KUKA KRL program: EPS_2_251112_SAMH04_A_20250918124117.src

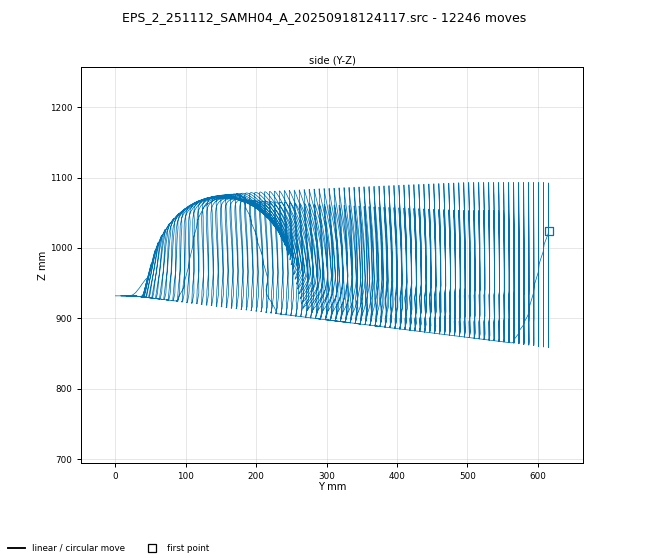
[picture p0: tool path of EPS_2_251112_SAMH04_A_20250918124117.src, 12246 of 12248 moves have a stored position in this frame; points joined in program order, loops and branches not executed]
&ACCESS RVP
&REL 4
&COMMENT QRS 19112012
&PARAM EDITMASK = *
DEF PART()
EXT BAS (BAS_COMMAND :IN,REAL :IN )
INT I
BAS (#INITMOV,0 )

;KUKA QRS Post kuka4.cps  Date:22-06-2017 !

File_ID=2836

QRS_PRE_INIT()

;Init var - Until changes are made in qrs_pre_init
Outlet_Square_prg=0
Inlet_1_Square_prg=0
Inlet_2_Square_prg=0
Inlet_3_Square_prg=0
Inlet_4_Square_prg=0
Inlet_5_Square_prg=0

Outlet_1={X 0.000, Y 497.840, Z 1018.000, B 0.000, E1 0.000 }
Inlet_1={X 0.000, Y 500.690, Z 978.000, B 0.000, E1 90.000 }
Outlet_1_type=150
Inlet_1_type=150
;QRS#1=Sidecore dimensions
;QRS#2=150-6" PVC SDR 28
;QRS#3=150-6" PVC SDR 28
;QRS#4=
;QRS#5=
;QRS#6=
;QRS#7=
;QRS#8=
;QRS#9=10-06 PSX
;QRS#10=10-06 PSX
;QRS#11=
;QRS#12=
;QRS#13=
;QRS#14=
;QRS#15=
;QRS#16=1220x127x1372 4,5'
;QRS#17=EPS Height
;QRS#18=1093
;QRS#19=*
;QRS#20= UPDATED VERSION 22-06-2017
;QRS#21=*
Outlet_Square=070
Inlet_1_Square=070
Inlet_2_Square=0
Inlet_3_Square=0
Inlet_4_Square=0
Inlet_5_Square=0
Mill_Square=1
Outlet_Square_Prg=203
Inlet_1_Square_prg=203

QRS_INIT()

$ADVANCE=5

; T1
PTP {E1 173.415,E2 173.415}
PTP {X 0,Y 615.497,A -85,B 0,C 180,E1 173.415,E2 173.415,E3 0,E4 0,E5 0,E6 0}
QRS_SPEED_INIT()
LIN {X 0,Y 615.497,Z 1023.816,A -85,B 0,C 180,E1 173.415,E2 173.415,E3 0,E4 0,E5 0,E6 0} C_VEL
LIN {X 0,Y 615.483,Z 1015.551,A -85,B 0,C 180,E1 172.702,E2 172.702} C_VEL
LIN {X 0,Y 615.494,Z 1005.669,A -85,B 0,C 180,E1 172.042,E2 172.042} C_VEL
LIN {X 0,Y 615.492,Z 997.912,A -85,B 0,C 180,E1 171.628,E2 171.628} C_VEL
LIN {X 0,Y 615.46,Z 989.058,A -85,B 0,C 180,E1 171.256,E2 171.256} C_VEL
LIN {X 0,Y 615.451,Z 979.837,A -85,B 0,C 180,E1 170.966,E2 170.966} C_VEL
LIN {X 0,Y 615.452,Z 970.156,A -85,B 0,C 180,E1 170.759,E2 170.759} C_VEL
LIN {X 0,Y 615.49,Z 894.306,A -85,B 0,C 180,E1 169.847,E2 169.847} C_VEL
LIN {X 0,Y 615.486,Z 880.811,A -85,B 0,C 180,E1 167.134,E2 167.134} C_VEL
LIN {X 0,Y 615.453,Z 867.509,A -85,B 0,C 180,E1 164.433,E2 164.433} C_VEL
LIN {X 0,Y 615.432,Z 858.511,A -85,B 0,C 180,E1 162.556,E2 162.556} C_VEL
LIN {X 0,Y 615.415,Z 858.509,A -85,B 0,C 180,E1 159.964,E2 159.964} C_VEL
LIN {X 0,Y 615.466,Z 858.507,A -85,B 0,C 180,E1 157.154,E2 157.154} C_VEL
LIN {X 0,Y 615.441,Z 858.511,A -85,B 0,C 180,E1 154.282,E2 154.282} C_VEL
LIN {X 0,Y 615.431,Z 858.511,A -85,B 0,C 180,E1 152.082,E2 152.082} C_VEL
LIN {X 0,Y 615.419,Z 858.51,A -85,B 0,C 180,E1 149.836,E2 149.836} C_VEL
LIN {X 0,Y 615.412,Z 858.51,A -85,B 0,C 180,E1 147.538,E2 147.538} C_VEL
LIN {X 0,Y 615.447,Z 858.511,A -85,B 0,C 180,E1 145.975,E2 145.975} C_VEL
LIN {X 0,Y 615.421,Z 858.51,A -85,B 0,C 180,E1 143.57,E2 143.57} C_VEL
LIN {X 0,Y 615.415,Z 858.509,A -85,B 0,C 180,E1 141.09,E2 141.09} C_VEL
LIN {X 0,Y 615.417,Z 858.508,A -85,B 0,C 180,E1 138.913,E2 138.913} C_VEL
LIN {X 0,Y 615.42,Z 858.508,A -85,B 0,C 180,E1 136.749,E2 136.749} C_VEL
LIN {X 0,Y 615.469,Z 858.506,A -85,B 0,C 180,E1 134.151,E2 134.151} C_VEL
LIN {X 0,Y 615.462,Z 858.513,A -85,B 0,C 180,E1 131.476,E2 131.476} C_VEL
LIN {X 0,Y 615.419,Z 858.51,A -85,B 0,C 180,E1 128.91,E2 128.91} C_VEL
LIN {X 0,Y 615.415,Z 858.509,A -85,B 0,C 180,E1 126.43,E2 126.43} C_VEL
LIN {X 0,Y 615.431,Z 858.508,A -85,B 0,C 180,E1 124.026,E2 124.026} C_VEL
LIN {X 0,Y 615.476,Z 858.512,A -85,B 0,C 180,E1 121.083,E2 121.083} C_VEL
LIN {X 0,Y 615.42,Z 858.51,A -85,B 0,C 180,E1 118.438,E2 118.438} C_VEL
LIN {X 0,Y 615.423,Z 858.511,A -85,B 0,C 180,E1 116.447,E2 116.447} C_VEL
LIN {X 0,Y 615.421,Z 858.51,A -85,B 0,C 180,E1 114.275,E2 114.275} C_VEL
LIN {X 0,Y 615.419,Z 858.51,A -85,B 0,C 180,E1 112.139,E2 112.139} C_VEL
LIN {X 0,Y 615.418,Z 858.51,A -85,B 0,C 180,E1 110.035,E2 110.035} C_VEL
LIN {X 0,Y 615.419,Z 858.51,A -85,B 0,C 180,E1 107.959,E2 107.959} C_VEL
LIN {X 0,Y 615.421,Z 858.51,A -85,B 0,C 180,E1 105.907,E2 105.907} C_VEL
LIN {X 0,Y 615.425,Z 858.51,A -85,B 0,C 180,E1 103.876,E2 103.876} C_VEL
LIN {X 0,Y 615.43,Z 858.511,A -85,B 0,C 180,E1 101.862,E2 101.862} C_VEL
LIN {X 0,Y 615.439,Z 858.511,A -85,B 0,C 180,E1 99.863,E2 99.863} C_VEL
LIN {X 0,Y 615.45,Z 858.511,A -85,B 0,C 180,E1 97.876,E2 97.876} C_VEL
LIN {X 0,Y 615.414,Z 858.51,A -85,B 0,C 180,E1 95.242,E2 95.242} C_VEL
LIN {X 0,Y 615.417,Z 858.51,A -85,B 0,C 180,E1 93.273,E2 93.273} C_VEL
LIN {X 0,Y 615.42,Z 858.511,A -85,B 0,C 180,E1 91.309,E2 91.309} C_VEL
LIN {X 0,Y 615.432,Z 858.511,A -85,B 0,C 180,E1 89.346,E2 89.346} C_VEL
LIN {X 0,Y 615.446,Z 858.511,A -85,B 0,C 180,E1 87.382,E2 87.382} C_VEL
LIN {X 0,Y 615.413,Z 858.51,A -85,B 0,C 180,E1 84.758,E2 84.758} C_VEL
LIN {X 0,Y 615.416,Z 858.51,A -85,B 0,C 180,E1 82.783,E2 82.783} C_VEL
LIN {X 0,Y 615.421,Z 858.51,A -85,B 0,C 180,E1 80.8,E2 80.8} C_VEL
LIN {X 0,Y 615.427,Z 858.511,A -85,B 0,C 180,E1 78.806,E2 78.806} C_VEL
LIN {X 0,Y 615.434,Z 858.511,A -85,B 0,C 180,E1 76.797,E2 76.797} C_VEL
LIN {X 0,Y 615.437,Z 858.512,A -85,B 0,C 180,E1 74.772,E2 74.772} C_VEL
LIN {X 0,Y 615.446,Z 858.511,A -85,B 0,C 180,E1 72.728,E2 72.728} C_VEL
LIN {X 0,Y 615.448,Z 858.511,A -85,B 0,C 180,E1 70.661,E2 70.661} C_VEL
LIN {X 0,Y 615.448,Z 858.511,A -85,B 0,C 180,E1 68.566,E2 68.566} C_VEL
LIN {X 0,Y 615.414,Z 858.51,A -85,B 0,C 180,E1 66.008,E2 66.008} C_VEL
LIN {X 0,Y 615.437,Z 858.511,A -85,B 0,C 180,E1 64.282,E2 64.282} C_VEL
LIN {X 0,Y 615.428,Z 858.511,A -85,B 0,C 180,E1 62.082,E2 62.082} C_VEL
LIN {X 0,Y 615.418,Z 858.51,A -85,B 0,C 180,E1 59.836,E2 59.836} C_VEL
LIN {X 0,Y 615.41,Z 858.51,A -85,B 0,C 180,E1 57.538,E2 57.538} C_VEL
LIN {X 0,Y 615.444,Z 858.511,A -85,B 0,C 180,E1 55.975,E2 55.975} C_VEL
LIN {X 0,Y 615.419,Z 858.51,A -85,B 0,C 180,E1 53.57,E2 53.57} C_VEL
LIN {X 0,Y 615.411,Z 858.51,A -85,B 0,C 180,E1 51.09,E2 51.09} C_VEL
LIN {X 0,Y 615.416,Z 858.509,A -85,B 0,C 180,E1 48.914,E2 48.914} C_VEL
LIN {X 0,Y 615.419,Z 858.509,A -85,B 0,C 180,E1 46.749,E2 46.749} C_VEL
LIN {X 0,Y 615.468,Z 858.507,A -85,B 0,C 180,E1 44.152,E2 44.152} C_VEL
LIN {X 0,Y 615.462,Z 858.512,A -85,B 0,C 180,E1 41.477,E2 41.477} C_VEL
LIN {X 0,Y 615.426,Z 858.511,A -85,B 0,C 180,E1 39.055,E2 39.055} C_VEL
LIN {X 0,Y 615.413,Z 858.509,A -85,B 0,C 180,E1 36.43,E2 36.43} C_VEL
LIN {X 0,Y 615.43,Z 858.508,A -85,B 0,C 180,E1 34.026,E2 34.026} C_VEL
LIN {X 0,Y 615.455,Z 858.508,A -85,B 0,C 180,E1 31.688,E2 31.688} C_VEL
LIN {X 0,Y 615.433,Z 858.511,A -85,B 0,C 180,E1 28.661,E2 28.661} C_VEL
LIN {X 0,Y 615.423,Z 858.511,A -85,B 0,C 180,E1 26.448,E2 26.448} C_VEL
LIN {X 0,Y 615.418,Z 858.51,A -85,B 0,C 180,E1 24.275,E2 24.275} C_VEL
LIN {X 0,Y 615.416,Z 858.51,A -85,B 0,C 180,E1 22.14,E2 22.14} C_VEL
LIN {X 0,Y 615.415,Z 858.511,A -85,B 0,C 180,E1 20.036,E2 20.036} C_VEL
LIN {X 0,Y 615.416,Z 858.51,A -85,B 0,C 180,E1 17.959,E2 17.959} C_VEL
LIN {X 0,Y 615.418,Z 858.51,A -85,B 0,C 180,E1 15.907,E2 15.907} C_VEL
LIN {X 0,Y 615.422,Z 858.511,A -85,B 0,C 180,E1 13.876,E2 13.876} C_VEL
LIN {X 0,Y 615.427,Z 858.511,A -85,B 0,C 180,E1 11.862,E2 11.862} C_VEL
LIN {X 0,Y 615.436,Z 858.511,A -85,B 0,C 180,E1 9.863,E2 9.863} C_VEL
LIN {X 0,Y 615.447,Z 858.511,A -85,B 0,C 180,E1 7.876,E2 7.876} C_VEL
LIN {X 0,Y 615.411,Z 858.51,A -85,B 0,C 180,E1 5.242,E2 5.242} C_VEL
LIN {X 0,Y 615.412,Z 858.511,A -85,B 0,C 180,E1 3.274,E2 3.274} C_VEL
LIN {X 0,Y 615.421,Z 858.511,A -85,B 0,C 180,E1 1.309,E2 1.309} C_VEL
LIN {X 0,Y 615.431,Z 858.511,A -85,B 0,C 180,E1 -0.654,E2 -0.654} C_VEL
LIN {X 0,Y 615.443,Z 858.511,A -85,B 0,C 180,E1 -2.618,E2 -2.618} C_VEL
LIN {X 0,Y 615.411,Z 858.51,A -85,B 0,C 180,E1 -5.242,E2 -5.242} C_VEL
LIN {X 0,Y 615.414,Z 858.51,A -85,B 0,C 180,E1 -7.216,E2 -7.216} C_VEL
LIN {X 0,Y 615.418,Z 858.511,A -85,B 0,C 180,E1 -9.2,E2 -9.2} C_VEL
LIN {X 0,Y 615.424,Z 858.511,A -85,B 0,C 180,E1 -11.194,E2 -11.194} C_VEL
LIN {X 0,Y 615.431,Z 858.511,A -85,B 0,C 180,E1 -13.202,E2 -13.202} C_VEL
LIN {X 0,Y 615.437,Z 858.511,A -85,B 0,C 180,E1 -15.227,E2 -15.227} C_VEL
LIN {X 0,Y 615.442,Z 858.511,A -85,B 0,C 180,E1 -17.272,E2 -17.272} C_VEL
LIN {X 0,Y 615.445,Z 858.512,A -85,B 0,C 180,E1 -19.339,E2 -19.339} C_VEL
LIN {X 0,Y 615.445,Z 858.512,A -85,B 0,C 180,E1 -21.433,E2 -21.433} C_VEL
LIN {X 0,Y 615.412,Z 858.51,A -85,B 0,C 180,E1 -23.992,E2 -23.992} C_VEL
LIN {X 0,Y 615.434,Z 858.511,A -85,B 0,C 180,E1 -25.718,E2 -25.718} C_VEL
LIN {X 0,Y 615.425,Z 858.511,A -85,B 0,C 180,E1 -27.918,E2 -27.918} C_VEL
LIN {X 0,Y 615.416,Z 858.511,A -85,B 0,C 180,E1 -30.164,E2 -30.164} C_VEL
LIN {X 0,Y 615.408,Z 858.51,A -85,B 0,C 180,E1 -32.462,E2 -32.462} C_VEL
LIN {X 0,Y 615.441,Z 858.511,A -85,B 0,C 180,E1 -34.025,E2 -34.025} C_VEL
LIN {X 0,Y 615.416,Z 858.511,A -85,B 0,C 180,E1 -36.429,E2 -36.429} C_VEL
LIN {X 0,Y 615.411,Z 858.51,A -85,B 0,C 180,E1 -38.91,E2 -38.91} C_VEL
LIN {X 0,Y 615.414,Z 858.509,A -85,B 0,C 180,E1 -41.086,E2 -41.086} C_VEL
LIN {X 0,Y 615.417,Z 858.509,A -85,B 0,C 180,E1 -43.251,E2 -43.251} C_VEL
LIN {X 0,Y 615.468,Z 858.508,A -85,B 0,C 180,E1 -45.848,E2 -45.848} C_VEL
LIN {X 0,Y 615.459,Z 858.512,A -85,B 0,C 180,E1 -48.523,E2 -48.523} C_VEL
LIN {X 0,Y 615.423,Z 858.511,A -85,B 0,C 180,E1 -50.945,E2 -50.945} C_VEL
LIN {X 0,Y 615.411,Z 858.51,A -85,B 0,C 180,E1 -53.57,E2 -53.57} C_VEL
LIN {X 0,Y 615.428,Z 858.509,A -85,B 0,C 180,E1 -55.974,E2 -55.974} C_VEL
LIN {X 0,Y 615.469,Z 858.512,A -85,B 0,C 180,E1 -58.917,E2 -58.917} C_VEL
LIN {X 0,Y 615.415,Z 858.511,A -85,B 0,C 180,E1 -61.562,E2 -61.562} C_VEL
LIN {X 0,Y 615.42,Z 858.511,A -85,B 0,C 180,E1 -63.553,E2 -63.553} C_VEL
LIN {X 0,Y 615.416,Z 858.511,A -85,B 0,C 180,E1 -65.725,E2 -65.725} C_VEL
LIN {X 0,Y 615.414,Z 858.511,A -85,B 0,C 180,E1 -67.861,E2 -67.861} C_VEL
LIN {X 0,Y 615.431,Z 858.559,A -85,B 0,C 180,E1 -68.566,E2 -68.566} C_VEL
LIN {X 0,Y 615.473,Z 876.687,A -85,B 0,C 180,E1 -71.399,E2 -71.399} C_VEL
LIN {X 0,Y 615.484,Z 894.205,A -85,B 0,C 180,E1 -74.095,E2 -74.095} C_VEL
LIN {X 0,Y 615.455,Z 912.003,A -85,B 0,C 180,E1 -76.798,E2 -76.798} C_VEL
LIN {X 0,Y 615.493,Z 930.889,A -85,B 0,C 180,E1 -79.639,E2 -79.639} C_VEL
LIN {X 0,Y 615.483,Z 932.416,A -85,B 0,C 180,E1 -79.868,E2 -79.868} C_VEL
LIN {X 0,Y 615.47,Z 1009.935,A -85,B 0,C 180,E1 -80.801,E2 -80.801} C_VEL
LIN {X 0,Y 615.465,Z 1019.696,A -85,B 0,C 180,E1 -81.008,E2 -81.008} C_VEL
LIN {X 0,Y 615.471,Z 1030.154,A -85,B 0,C 180,E1 -81.339,E2 -81.339} C_VEL
LIN {X 0,Y 615.497,Z 1040.424,A -85,B 0,C 180,E1 -81.794,E2 -81.794} C_VEL
LIN {X 0,Y 615.477,Z 1050.199,A -85,B 0,C 180,E1 -82.372,E2 -82.372} C_VEL
LIN {X 0,Y 615.493,Z 1057.933,A -85,B 0,C 180,E1 -82.942,E2 -82.942} C_VEL
LIN {X 0,Y 615.497,Z 1065.332,A -85,B 0,C 180,E1 -83.608,E2 -83.608} C_VEL
LIN {X 0,Y 615.498,Z 1072.736,A -85,B 0,C 180,E1 -84.43,E2 -84.43} C_VEL
LIN {X 0,Y 615.497,Z 1078.532,A -85,B 0,C 180,E1 -85.251,E2 -85.251} C_VEL
LIN {X 0,Y 615.493,Z 1083.1,A -85,B 0,C 180,E1 -86.071,E2 -86.071} C_VEL
LIN {X 0,Y 615.493,Z 1086.068,A -85,B 0,C 180,E1 -86.727,E2 -86.727} C_VEL
LIN {X 0,Y 615.494,Z 1088.356,A -85,B 0,C 180,E1 -87.382,E2 -87.382} C_VEL
LIN {X 0,Y 615.499,Z 1090.085,A -85,B 0,C 180,E1 -88.037,E2 -88.037} C_VEL
LIN {X 0,Y 615.493,Z 1091.33,A -85,B 0,C 180,E1 -88.691,E2 -88.691} C_VEL
LIN {X 0,Y 615.491,Z 1092.104,A -85,B 0,C 180,E1 -89.346,E2 -89.346} C_VEL
LIN {X 0,Y 615.491,Z 1092.389,A -85,B 0,C 180,E1 -90,E2 -90} C_VEL
LIN {X 0,Y 615.491,Z 1092.104,A -85,B 0,C 180,E1 -90.654,E2 -90.654} C_VEL
LIN {X 0,Y 615.493,Z 1091.33,A -85,B 0,C 180,E1 -91.308,E2 -91.308} C_VEL
LIN {X 0,Y 615.499,Z 1090.085,A -85,B 0,C 180,E1 -91.963,E2 -91.963} C_VEL
LIN {X 0,Y 615.488,Z 1087.221,A -85,B 0,C 180,E1 -92.945,E2 -92.945} C_VEL
LIN {X 0,Y 615.492,Z 1084.604,A -85,B 0,C 180,E1 -93.601,E2 -93.601} C_VEL
LIN {X 0,Y 615.496,Z 1079.483,A -85,B 0,C 180,E1 -94.584,E2 -94.584} C_VEL
LIN {X 0,Y 615.495,Z 1073.969,A -85,B 0,C 180,E1 -95.405,E2 -95.405} C_VEL
LIN {X 0,Y 615.498,Z 1067.019,A -85,B 0,C 180,E1 -96.227,E2 -96.227} C_VEL
LIN {X 0,Y 615.495,Z 1059.859,A -85,B 0,C 180,E1 -96.901,E2 -96.901} C_VEL
LIN {X 0,Y 615.477,Z 1052.626,A -85,B 0,C 180,E1 -97.463,E2 -97.463} C_VEL
LIN {X 0,Y 615.494,Z 1044.87,A -85,B 0,C 180,E1 -97.958,E2 -97.958} C_VEL
LIN {X 0,Y 615.493,Z 1036.916,A -85,B 0,C 180,E1 -98.371,E2 -98.371} C_VEL
LIN {X 0,Y 615.471,Z 1027.764,A -85,B 0,C 180,E1 -98.744,E2 -98.744} C_VEL
LIN {X 0,Y 615.465,Z 1019.706,A -85,B 0,C 180,E1 -98.992,E2 -98.992} C_VEL
LIN {X 0,Y 615.47,Z 1009.951,A -85,B 0,C 180,E1 -99.199,E2 -99.199} C_VEL
LIN {X 0,Y 615.483,Z 932.418,A -85,B 0,C 180,E1 -100.132,E2 -100.132} C_VEL
LIN {X 0,Y 615.485,Z 914.226,A -85,B 0,C 180,E1 -102.865,E2 -102.865} C_VEL
LIN {X 0,Y 615.459,Z 896.439,A -85,B 0,C 180,E1 -105.566,E2 -105.566} C_VEL
LIN {X 0,Y 615.463,Z 879.807,A -85,B 0,C 180,E1 -108.118,E2 -108.118} C_VEL
LIN {X 0,Y 615.494,Z 861.903,A -85,B 0,C 180,E1 -110.905,E2 -110.905} C_VEL
LIN {X 0,Y 615.427,Z 858.509,A -85,B 0,C 180,E1 -111.478,E2 -111.478} C_VEL
LIN {X 0,Y 615.428,Z 858.509,A -85,B 0,C 180,E1 -113.559,E2 -113.559} C_VEL
LIN {X 0,Y 615.423,Z 858.509,A -85,B 0,C 180,E1 -115.719,E2 -115.719} C_VEL
LIN {X 0,Y 615.416,Z 858.51,A -85,B 0,C 180,E1 -117.919,E2 -117.919} C_VEL
LIN {X 0,Y 615.41,Z 858.51,A -85,B 0,C 180,E1 -120.164,E2 -120.164} C_VEL
LIN {X 0,Y 615.409,Z 858.51,A -85,B 0,C 180,E1 -122.462,E2 -122.462} C_VEL
LIN {X 0,Y 615.412,Z 858.511,A -85,B 0,C 180,E1 -124.691,E2 -124.691} C_VEL
LIN {X 0,Y 615.42,Z 858.511,A -85,B 0,C 180,E1 -126.928,E2 -126.928} C_VEL
LIN {X 0,Y 615.496,Z 858.51,A -85,B 0,C 180,E1 -129.749,E2 -129.749} C_VEL
LIN {X 0,Y 615.431,Z 858.509,A -85,B 0,C 180,E1 -132.358,E2 -132.358} C_VEL
LIN {X 0,Y 615.468,Z 858.509,A -85,B 0,C 180,E1 -134.151,E2 -134.151} C_VEL
LIN {X 0,Y 615.416,Z 858.51,A -85,B 0,C 180,E1 -136.749,E2 -136.749} C_VEL
LIN {X 0,Y 615.412,Z 858.51,A -85,B 0,C 180,E1 -138.914,E2 -138.914} C_VEL
LIN {X 0,Y 615.409,Z 858.51,A -85,B 0,C 180,E1 -141.09,E2 -141.09} C_VEL
LIN {X 0,Y 615.413,Z 858.511,A -85,B 0,C 180,E1 -143.57,E2 -143.57} C_VEL
LIN {X 0,Y 615.436,Z 858.512,A -85,B 0,C 180,E1 -145.975,E2 -145.975} C_VEL
LIN {X 0,Y 615.451,Z 858.509,A -85,B 0,C 180,E1 -148.92,E2 -148.92} C_VEL
LIN {X 0,Y 615.419,Z 858.51,A -85,B 0,C 180,E1 -151.339,E2 -151.339} C_VEL
LIN {X 0,Y 615.412,Z 858.51,A -85,B 0,C 180,E1 -153.553,E2 -153.553} C_VEL
LIN {X 0,Y 615.409,Z 858.51,A -85,B 0,C 180,E1 -155.725,E2 -155.725} C_VEL
LIN {X 0,Y 615.408,Z 858.51,A -85,B 0,C 180,E1 -157.861,E2 -157.861} C_VEL
LIN {X 0,Y 615.407,Z 858.51,A -85,B 0,C 180,E1 -159.965,E2 -159.965} C_VEL
LIN {X 0,Y 615.411,Z 858.511,A -85,B 0,C 180,E1 -162.385,E2 -162.385} C_VEL
LIN {X 0,Y 615.436,Z 858.756,A -85,B 0,C 180,E1 -162.728,E2 -162.728} C_VEL
LIN {X 0,Y 615.483,Z 872.058,A -85,B 0,C 180,E1 -165.451,E2 -165.451} C_VEL
LIN {X 0,Y 615.476,Z 885.351,A -85,B 0,C 180,E1 -168.139,E2 -168.139} C_VEL
LIN {X 0,Y 615.487,Z 894.569,A -85,B 0,C 180,E1 -169.951,E2 -169.951} C_VEL
LIN {X 0,Y 615.459,Z 969.743,A -85,B 0,C 180,E1 -170.842,E2 -170.842} C_VEL
LIN {X 0,Y 615.458,Z 977.917,A -85,B 0,C 180,E1 -171.008,E2 -171.008} C_VEL
LIN {X 0,Y 615.464,Z 986.468,A -85,B 0,C 180,E1 -171.257,E2 -171.257} C_VEL
LIN {X 0,Y 615.483,Z 994.071,A -85,B 0,C 180,E1 -171.546,E2 -171.546} C_VEL
LIN {X 0,Y 615.497,Z 1002.587,A -85,B 0,C 180,E1 -171.96,E2 -171.96} C_VEL
LIN {X 0,Y 615.479,Z 1010.755,A -85,B 0,C 180,E1 -172.455,E2 -172.455} C_VEL
LIN {X 0,Y 615.49,Z 1017.392,A -85,B 0,C 180,E1 -172.942,E2 -172.942} C_VEL
LIN {X 0,Y 615.498,Z 1023.187,A -85,B 0,C 180,E1 -173.444,E2 -173.444} C_VEL
LIN {X 0,Y 615.499,Z 1029.537,A -85,B 0,C 180,E1 -174.102,E2 -174.102} C_VEL
LIN {X 0,Y 615.495,Z 1035.986,A -85,B 0,C 180,E1 -174.923,E2 -174.923} C_VEL
LIN {X 0,Y 615.492,Z 1041.124,A -85,B 0,C 180,E1 -175.744,E2 -175.744} C_VEL
LIN {X 0,Y 615.493,Z 1045.888,A -85,B 0,C 180,E1 -176.727,E2 -176.727} C_VEL
LIN {X 0,Y 615.493,Z 1048.201,A -85,B 0,C 180,E1 -177.382,E2 -177.382} C_VEL
LIN {X 0,Y 615.498,Z 1049.977,A -85,B 0,C 180,E1 -178.037,E2 -178.037} C_VEL
LIN {X 0,Y 615.492,Z 1051.267,A -85,B 0,C 180,E1 -178.692,E2 -178.692} C_VEL
LIN {X 0,Y 615.491,Z 1052.084,A -85,B 0,C 180,E1 -179.346,E2 -179.346} C_VEL
LIN {X 0,Y 615.492,Z 1052.385,A -85,B 0,C 180,E1 -180,E2 -180} C_VEL
LIN {X 0,Y 615.492,Z 1052.125,A -85,B 0,C 180,E1 -180.655,E2 -180.655} C_VEL
LIN {X 0,Y 615.494,Z 1051.393,A -85,B 0,C 180,E1 -181.309,E2 -181.309} C_VEL
LIN {X 0,Y 615.499,Z 1050.193,A -85,B 0,C 180,E1 -181.963,E2 -181.963} C_VEL
LIN {X 0,Y 615.49,Z 1047.375,A -85,B 0,C 180,E1 -182.946,E2 -182.946} C_VEL
LIN {X 0,Y 615.491,Z 1044.809,A -85,B 0,C 180,E1 -183.601,E2 -183.601} C_VEL
LIN {X 0,Y 615.495,Z 1039.741,A -85,B 0,C 180,E1 -184.585,E2 -184.585} C_VEL
LIN {X 0,Y 615.496,Z 1034.285,A -85,B 0,C 180,E1 -185.406,E2 -185.406} C_VEL
LIN {X 0,Y 615.497,Z 1027.45,A -85,B 0,C 180,E1 -186.228,E2 -186.228} C_VEL
LIN {X 0,Y 615.497,Z 1023.816,A -85,B 0,C 180,E1 -186.585,E2 -186.585} C_VEL
LIN {X 0,Y 614.845,Z 1019.734,A -85,B 0,C 180,E1 -186.977,E2 -186.977} C_VEL
LIN {X 0,Y 612.024,Z 1012.698,A -85,B 0,C 180,E1 -187.582,E2 -187.582} C_VEL
LIN {X 0,Y 609.189,Z 1005.072,A -85,B 0,C 180,E1 -188.113,E2 -188.113} C_VEL
LIN {X 0,Y 608.503,Z 999.979,A -85,B 0,C 180,E1 -188.386,E2 -188.386} C_VEL
LIN {X 0,Y 608.451,Z 989.374,A -85,B 0,C 180,E1 -188.846,E2 -188.846} C_VEL
LIN {X 0,Y 608.474,Z 979.354,A -85,B 0,C 180,E1 -189.159,E2 -189.159} C_VEL
LIN {X 0,Y 608.459,Z 970.614,A -85,B 0,C 180,E1 -189.348,E2 -189.348} C_VEL
LIN {X 0,Y 608.532,Z 922.356,A -85,B 0,C 180,E1 -189.934,E2 -189.934} C_VEL
LIN {X 0,Y 608.449,Z 894.624,A -85,B 0,C 180,E1 -190.272,E2 -190.272} C_VEL
LIN {X 0,Y 608.455,Z 881.046,A -85,B 0,C 180,E1 -193.017,E2 -193.017} C_VEL
LIN {X 0,Y 608.423,Z 867.676,A -85,B 0,C 180,E1 -195.751,E2 -195.751} C_VEL
LIN {X 0,Y 608.41,Z 859.507,A -85,B 0,C 180,E1 -197.478,E2 -197.478} C_VEL
LIN {X 0,Y 608.409,Z 859.506,A -85,B 0,C 180,E1 -199.572,E2 -199.572} C_VEL
LIN {X 0,Y 608.424,Z 859.504,A -85,B 0,C 180,E1 -201.694,E2 -201.694} C_VEL
LIN {X 0,Y 608.418,Z 859.504,A -85,B 0,C 180,E1 -204.573,E2 -204.573} C_VEL
LIN {X 0,Y 608.427,Z 859.511,A -85,B 0,C 180,E1 -207.52,E2 -207.52} C_VEL
LIN {X 0,Y 608.409,Z 859.507,A -85,B 0,C 180,E1 -209.962,E2 -209.962} C_VEL
LIN {X 0,Y 608.4,Z 859.505,A -85,B 0,C 180,E1 -212.513,E2 -212.513} C_VEL
LIN {X 0,Y 608.392,Z 859.506,A -85,B 0,C 180,E1 -214.898,E2 -214.898} C_VEL
LIN {X 0,Y 608.428,Z 859.503,A -85,B 0,C 180,E1 -217.153,E2 -217.153} C_VEL
LIN {X 0,Y 608.436,Z 859.505,A -85,B 0,C 180,E1 -220.327,E2 -220.327} C_VEL
LIN {X 0,Y 608.426,Z 859.508,A -85,B 0,C 180,E1 -222.331,E2 -222.331} C_VEL
LIN {X 0,Y 608.4,Z 859.507,A -85,B 0,C 180,E1 -224.802,E2 -224.802} C_VEL
LIN {X 0,Y 608.388,Z 859.507,A -85,B 0,C 180,E1 -227.034,E2 -227.034} C_VEL
LIN {X 0,Y 608.42,Z 859.504,A -85,B 0,C 180,E1 -229.694,E2 -229.694} C_VEL
LIN {X 0,Y 608.442,Z 859.505,A -85,B 0,C 180,E1 -232.846,E2 -232.846} C_VEL
LIN {X 0,Y 608.413,Z 859.503,A -85,B 0,C 180,E1 -235.527,E2 -235.527} C_VEL
LIN {X 0,Y 608.412,Z 859.504,A -85,B 0,C 180,E1 -237.902,E2 -237.902} C_VEL
LIN {X 0,Y 608.422,Z 859.504,A -85,B 0,C 180,E1 -240.218,E2 -240.218} C_VEL
LIN {X 0,Y 608.462,Z 859.506,A -85,B 0,C 180,E1 -242.797,E2 -242.797} C_VEL
LIN {X 0,Y 608.426,Z 859.507,A -85,B 0,C 180,E1 -245.428,E2 -245.428} C_VEL
LIN {X 0,Y 608.42,Z 859.506,A -85,B 0,C 180,E1 -247.593,E2 -247.593} C_VEL
LIN {X 0,Y 608.42,Z 859.506,A -85,B 0,C 180,E1 -249.724,E2 -249.724} C_VEL
LIN {X 0,Y 608.404,Z 859.508,A -85,B 0,C 180,E1 -251.827,E2 -251.827} C_VEL
LIN {X 0,Y 608.417,Z 859.506,A -85,B 0,C 180,E1 -253.905,E2 -253.905} C_VEL
LIN {X 0,Y 608.405,Z 859.504,A -85,B 0,C 180,E1 -256.642,E2 -256.642} C_VEL
LIN {X 0,Y 608.449,Z 859.505,A -85,B 0,C 180,E1 -259.35,E2 -259.35} C_VEL
LIN {X 0,Y 608.419,Z 859.51,A -85,B 0,C 180,E1 -262.032,E2 -262.032} C_VEL
LIN {X 0,Y 608.402,Z 859.505,A -85,B 0,C 180,E1 -264.698,E2 -264.698} C_VEL
LIN {X 0,Y 608.427,Z 859.503,A -85,B 0,C 180,E1 -267.352,E2 -267.352} C_VEL
LIN {X 0,Y 608.477,Z 859.505,A -85,B 0,C 180,E1 -270,E2 -270} C_VEL
LIN {X 0,Y 608.44,Z 859.505,A -85,B 0,C 180,E1 -272.648,E2 -272.648} C_VEL
LIN {X 0,Y 608.4,Z 859.505,A -85,B 0,C 180,E1 -275.303,E2 -275.303} C_VEL
LIN {X 0,Y 608.4,Z 859.505,A -85,B 0,C 180,E1 -277.3,E2 -277.3} C_VEL
LIN {X 0,Y 608.411,Z 859.504,A -85,B 0,C 180,E1 -279.307,E2 -279.307} C_VEL
LIN {X 0,Y 608.406,Z 859.506,A -85,B 0,C 180,E1 -281.325,E2 -281.325} C_VEL
LIN {X 0,Y 608.411,Z 859.505,A -85,B 0,C 180,E1 -283.358,E2 -283.358} C_VEL
LIN {X 0,Y 608.406,Z 859.505,A -85,B 0,C 180,E1 -286.096,E2 -286.096} C_VEL
LIN {X 0,Y 608.442,Z 859.51,A -85,B 0,C 180,E1 -288.87,E2 -288.87} C_VEL
LIN {X 0,Y 608.422,Z 859.504,A -85,B 0,C 180,E1 -291.694,E2 -291.694} C_VEL
LIN {X 0,Y 608.417,Z 859.504,A -85,B 0,C 180,E1 -294.573,E2 -294.573} C_VEL
LIN {X 0,Y 608.426,Z 859.511,A -85,B 0,C 180,E1 -297.519,E2 -297.519} C_VEL
LIN {X 0,Y 608.409,Z 859.507,A -85,B 0,C 180,E1 -299.961,E2 -299.961} C_VEL
LIN {X 0,Y 608.399,Z 859.505,A -85,B 0,C 180,E1 -302.512,E2 -302.512} C_VEL
LIN {X 0,Y 608.39,Z 859.507,A -85,B 0,C 180,E1 -304.897,E2 -304.897} C_VEL
LIN {X 0,Y 608.427,Z 859.503,A -85,B 0,C 180,E1 -307.152,E2 -307.152} C_VEL
LIN {X 0,Y 608.438,Z 859.505,A -85,B 0,C 180,E1 -310.327,E2 -310.327} C_VEL
LIN {X 0,Y 608.423,Z 859.508,A -85,B 0,C 180,E1 -312.33,E2 -312.33} C_VEL
LIN {X 0,Y 608.399,Z 859.506,A -85,B 0,C 180,E1 -314.802,E2 -314.802} C_VEL
LIN {X 0,Y 608.387,Z 859.507,A -85,B 0,C 180,E1 -317.034,E2 -317.034} C_VEL
LIN {X 0,Y 608.421,Z 859.504,A -85,B 0,C 180,E1 -319.694,E2 -319.694} C_VEL
LIN {X 0,Y 608.439,Z 859.505,A -85,B 0,C 180,E1 -322.846,E2 -322.846} C_VEL
LIN {X 0,Y 608.411,Z 859.504,A -85,B 0,C 180,E1 -325.526,E2 -325.526} C_VEL
LIN {X 0,Y 608.412,Z 859.504,A -85,B 0,C 180,E1 -327.902,E2 -327.902} C_VEL
LIN {X 0,Y 608.42,Z 859.504,A -85,B 0,C 180,E1 -330.217,E2 -330.217} C_VEL
LIN {X 0,Y 608.426,Z 859.508,A -85,B 0,C 180,E1 -333.224,E2 -333.224} C_VEL
LIN {X 0,Y 608.393,Z 859.506,A -85,B 0,C 180,E1 -335.866,E2 -335.866} C_VEL
LIN {X 0,Y 608.414,Z 859.503,A -85,B 0,C 180,E1 -338.306,E2 -338.306} C_VEL
LIN {X 0,Y 608.444,Z 859.508,A -85,B 0,C 180,E1 -341.13,E2 -341.13} C_VEL
LIN {X 0,Y 608.415,Z 859.506,A -85,B 0,C 180,E1 -343.905,E2 -343.905} C_VEL
LIN {X 0,Y 608.403,Z 859.505,A -85,B 0,C 180,E1 -346.642,E2 -346.642} C_VEL
LIN {X 0,Y 608.449,Z 859.505,A -85,B 0,C 180,E1 -349.35,E2 -349.35} C_VEL
LIN {X 0,Y 608.417,Z 859.51,A -85,B 0,C 180,E1 -352.032,E2 -352.032} C_VEL
LIN {X 0,Y 608.4,Z 859.505,A -85,B 0,C 180,E1 -354.697,E2 -354.697} C_VEL
LIN {X 0,Y 608.425,Z 859.503,A -85,B 0,C 180,E1 -357.351,E2 -357.351} C_VEL
LIN {X 0,Y 608.475,Z 859.505,A -85,B 0,C 180,E1 -360,E2 -360} C_VEL
LIN {X 0,Y 608.437,Z 859.505,A -85,B 0,C 180,E1 -362.648,E2 -362.648} C_VEL
LIN {X 0,Y 608.398,Z 859.505,A -85,B 0,C 180,E1 -365.302,E2 -365.302} C_VEL
LIN {X 0,Y 608.398,Z 859.505,A -85,B 0,C 180,E1 -367.3,E2 -367.3} C_VEL
LIN {X 0,Y 608.408,Z 859.505,A -85,B 0,C 180,E1 -369.306,E2 -369.306} C_VEL
LIN {X 0,Y 608.403,Z 859.506,A -85,B 0,C 180,E1 -371.325,E2 -371.325} C_VEL
LIN {X 0,Y 608.408,Z 859.506,A -85,B 0,C 180,E1 -373.357,E2 -373.357} C_VEL
LIN {X 0,Y 608.405,Z 859.505,A -85,B 0,C 180,E1 -376.095,E2 -376.095} C_VEL
LIN {X 0,Y 608.44,Z 859.51,A -85,B 0,C 180,E1 -378.87,E2 -378.87} C_VEL
LIN {X 0,Y 608.419,Z 859.505,A -85,B 0,C 180,E1 -381.693,E2 -381.693} C_VEL
LIN {X 0,Y 608.416,Z 859.505,A -85,B 0,C 180,E1 -384.572,E2 -384.572} C_VEL
LIN {X 0,Y 608.423,Z 859.511,A -85,B 0,C 180,E1 -387.519,E2 -387.519} C_VEL
LIN {X 0,Y 608.406,Z 859.507,A -85,B 0,C 180,E1 -389.961,E2 -389.961} C_VEL
LIN {X 0,Y 608.397,Z 859.505,A -85,B 0,C 180,E1 -392.512,E2 -392.512} C_VEL
LIN {X 0,Y 608.389,Z 859.507,A -85,B 0,C 180,E1 -394.897,E2 -394.897} C_VEL
LIN {X 0,Y 608.426,Z 859.504,A -85,B 0,C 180,E1 -397.152,E2 -397.152} C_VEL
LIN {X 0,Y 608.434,Z 859.505,A -85,B 0,C 180,E1 -400.327,E2 -400.327} C_VEL
LIN {X 0,Y 608.42,Z 859.508,A -85,B 0,C 180,E1 -402.33,E2 -402.33} C_VEL
LIN {X 0,Y 608.397,Z 859.507,A -85,B 0,C 180,E1 -404.801,E2 -404.801} C_VEL
LIN {X 0,Y 608.384,Z 859.507,A -85,B 0,C 180,E1 -407.034,E2 -407.034} C_VEL
LIN {X 0,Y 608.417,Z 859.505,A -85,B 0,C 180,E1 -409.693,E2 -409.693} C_VEL
LIN {X 0,Y 608.436,Z 859.505,A -85,B 0,C 180,E1 -412.846,E2 -412.846} C_VEL
LIN {X 0,Y 608.408,Z 859.504,A -85,B 0,C 180,E1 -415.526,E2 -415.526} C_VEL
LIN {X 0,Y 608.41,Z 859.504,A -85,B 0,C 180,E1 -417.902,E2 -417.902} C_VEL
LIN {X 0,Y 608.42,Z 859.505,A -85,B 0,C 180,E1 -420.218,E2 -420.218} C_VEL
LIN {X 0,Y 608.422,Z 859.508,A -85,B 0,C 180,E1 -423.224,E2 -423.224} C_VEL
LIN {X 0,Y 608.391,Z 859.507,A -85,B 0,C 180,E1 -425.866,E2 -425.866} C_VEL
LIN {X 0,Y 608.442,Z 859.688,A -85,B 0,C 180,E1 -428.485,E2 -428.485} C_VEL
LIN {X 0,Y 608.512,Z 876.436,A -85,B 0,C 180,E1 -431.132,E2 -431.132} C_VEL
LIN {X 0,Y 608.489,Z 894.302,A -85,B 0,C 180,E1 -433.907,E2 -433.907} C_VEL
LIN {X 0,Y 608.433,Z 912.167,A -85,B 0,C 180,E1 -436.643,E2 -436.643} C_VEL
LIN {X 0,Y 608.472,Z 931.149,A -85,B 0,C 180,E1 -439.518,E2 -439.518} C_VEL
LIN {X 0,Y 608.471,Z 932.684,A -85,B 0,C 180,E1 -439.75,E2 -439.75} C_VEL
LIN {X 0,Y 608.492,Z 1010.433,A -85,B 0,C 180,E1 -440.694,E2 -440.694} C_VEL
LIN {X 0,Y 608.492,Z 1020.068,A -85,B 0,C 180,E1 -440.904,E2 -440.904} C_VEL
LIN {X 0,Y 608.479,Z 1031.613,A -85,B 0,C 180,E1 -441.28,E2 -441.28} C_VEL
LIN {X 0,Y 608.478,Z 1042.229,A -85,B 0,C 180,E1 -441.782,E2 -441.782} C_VEL
LIN {X 0,Y 608.458,Z 1050.539,A -85,B 0,C 180,E1 -442.283,E2 -442.283} C_VEL
LIN {X 0,Y 608.459,Z 1058.399,A -85,B 0,C 180,E1 -442.867,E2 -442.867} C_VEL
LIN {X 0,Y 608.466,Z 1065.355,A -85,B 0,C 180,E1 -443.496,E2 -443.496} C_VEL
LIN {X 0,Y 608.469,Z 1073.19,A -85,B 0,C 180,E1 -444.366,E2 -444.366} C_VEL
LIN {X 0,Y 608.448,Z 1079.026,A -85,B 0,C 180,E1 -445.196,E2 -445.196} C_VEL
LIN {X 0,Y 608.431,Z 1083.63,A -85,B 0,C 180,E1 -446.026,E2 -446.026} C_VEL
LIN {X 0,Y 608.425,Z 1086.621,A -85,B 0,C 180,E1 -446.689,E2 -446.689} C_VEL
LIN {X 0,Y 608.423,Z 1088.93,A -85,B 0,C 180,E1 -447.352,E2 -447.352} C_VEL
LIN {X 0,Y 608.443,Z 1090.678,A -85,B 0,C 180,E1 -448.014,E2 -448.014} C_VEL
LIN {X 0,Y 608.445,Z 1091.933,A -85,B 0,C 180,E1 -448.676,E2 -448.676} C_VEL
LIN {X 0,Y 608.434,Z 1092.714,A -85,B 0,C 180,E1 -449.338,E2 -449.338} C_VEL
LIN {X 0,Y 608.431,Z 1093,A -85,B 0,C 180,E1 -450,E2 -450} C_VEL
LIN {X 0,Y 608.434,Z 1092.714,A -85,B 0,C 180,E1 -450.662,E2 -450.662} C_VEL
LIN {X 0,Y 608.445,Z 1091.934,A -85,B 0,C 180,E1 -451.324,E2 -451.324} C_VEL
LIN {X 0,Y 608.443,Z 1090.678,A -85,B 0,C 180,E1 -451.986,E2 -451.986} C_VEL
LIN {X 0,Y 608.444,Z 1087.786,A -85,B 0,C 180,E1 -452.979,E2 -452.979} C_VEL
LIN {X 0,Y 608.446,Z 1085.147,A -85,B 0,C 180,E1 -453.642,E2 -453.642} C_VEL
LIN {X 0,Y 608.447,Z 1079.985,A -85,B 0,C 180,E1 -454.638,E2 -454.638} C_VEL
LIN {X 0,Y 608.46,Z 1074.43,A -85,B 0,C 180,E1 -455.468,E2 -455.468} C_VEL
LIN {X 0,Y 608.455,Z 1066.669,A -85,B 0,C 180,E1 -456.376,E2 -456.376} C_VEL
LIN {X 0,Y 608.452,Z 1059.416,A -85,B 0,C 180,E1 -457.049,E2 -457.049} C_VEL
LIN {X 0,Y 608.458,Z 1051.761,A -85,B 0,C 180,E1 -457.633,E2 -457.633} C_VEL
LIN {X 0,Y 608.496,Z 1043.72,A -85,B 0,C 180,E1 -458.134,E2 -458.134} C_VEL
LIN {X 0,Y 608.486,Z 1035.39,A -85,B 0,C 180,E1 -458.552,E2 -458.552} C_VEL
LIN {X 0,Y 608.461,Z 1026.89,A -85,B 0,C 180,E1 -458.887,E2 -458.887} C_VEL
LIN {X 0,Y 608.49,Z 1017.587,A -85,B 0,C 180,E1 -459.159,E2 -459.159} C_VEL
LIN {X 0,Y 608.48,Z 1007.851,A -85,B 0,C 180,E1 -459.347,E2 -459.347} C_VEL
LIN {X 0,Y 608.471,Z 932.686,A -85,B 0,C 180,E1 -460.25,E2 -460.25} C_VEL
LIN {X 0,Y 608.452,Z 913.285,A -85,B 0,C 180,E1 -463.187,E2 -463.187} C_VEL
LIN {X 0,Y 608.491,Z 895.42,A -85,B 0,C 180,E1 -465.921,E2 -465.921} C_VEL
LIN {X 0,Y 608.506,Z 877.346,A -85,B 0,C 180,E1 -468.726,E2 -468.726} C_VEL
LIN {X 0,Y 608.504,Z 860.806,A -85,B 0,C 180,E1 -471.335,E2 -471.335} C_VEL
LIN {X 0,Y 608.412,Z 859.506,A -85,B 0,C 180,E1 -471.56,E2 -471.56} C_VEL
LIN {X 0,Y 608.39,Z 859.507,A -85,B 0,C 180,E1 -474.134,E2 -474.134} C_VEL
LIN {X 0,Y 608.422,Z 859.508,A -85,B 0,C 180,E1 -476.776,E2 -476.776} C_VEL
LIN {X 0,Y 608.419,Z 859.505,A -85,B 0,C 180,E1 -479.782,E2 -479.782} C_VEL
LIN {X 0,Y 608.41,Z 859.504,A -85,B 0,C 180,E1 -482.098,E2 -482.098} C_VEL
LIN {X 0,Y 608.407,Z 859.504,A -85,B 0,C 180,E1 -484.473,E2 -484.473} C_VEL
LIN {X 0,Y 608.434,Z 859.505,A -85,B 0,C 180,E1 -487.154,E2 -487.154} C_VEL
LIN {X 0,Y 608.415,Z 859.505,A -85,B 0,C 180,E1 -490.306,E2 -490.306} C_VEL
LIN {X 0,Y 608.382,Z 859.508,A -85,B 0,C 180,E1 -492.966,E2 -492.966} C_VEL
LIN {X 0,Y 608.394,Z 859.507,A -85,B 0,C 180,E1 -495.199,E2 -495.199} C_VEL
LIN {X 0,Y 608.456,Z 859.508,A -85,B 0,C 180,E1 -497.938,E2 -497.938} C_VEL
LIN {X 0,Y 608.407,Z 859.507,A -85,B 0,C 180,E1 -500.71,E2 -500.71} C_VEL
LIN {X 0,Y 608.384,Z 859.507,A -85,B 0,C 180,E1 -503.08,E2 -503.08} C_VEL
LIN {X 0,Y 608.407,Z 859.504,A -85,B 0,C 180,E1 -505.527,E2 -505.527} C_VEL
LIN {X 0,Y 608.414,Z 859.505,A -85,B 0,C 180,E1 -507.903,E2 -507.903} C_VEL
LIN {X 0,Y 608.427,Z 859.507,A -85,B 0,C 180,E1 -510.218,E2 -510.218} C_VEL
LIN {X 0,Y 608.408,Z 859.507,A -85,B 0,C 180,E1 -513.224,E2 -513.224} C_VEL
LIN {X 0,Y 608.388,Z 859.507,A -85,B 0,C 180,E1 -515.867,E2 -515.867} C_VEL
LIN {X 0,Y 608.414,Z 859.505,A -85,B 0,C 180,E1 -518.307,E2 -518.307} C_VEL
LIN {X 0,Y 608.457,Z 859.506,A -85,B 0,C 180,E1 -521.288,E2 -521.288} C_VEL
LIN {X 0,Y 608.409,Z 859.515,A -85,B 0,C 180,E1 -522.652,E2 -522.652} C_VEL
LIN {X 0,Y 608.454,Z 873.924,A -85,B 0,C 180,E1 -525.621,E2 -525.621} C_VEL
LIN {X 0,Y 608.433,Z 887.289,A -85,B 0,C 180,E1 -528.338,E2 -528.338} C_VEL
LIN {X 0,Y 608.44,Z 894.598,A -85,B 0,C 180,E1 -529.813,E2 -529.813} C_VEL
LIN {X 0,Y 608.481,Z 970.269,A -85,B 0,C 180,E1 -530.737,E2 -530.737} C_VEL
LIN {X 0,Y 608.477,Z 979.963,A -85,B 0,C 180,E1 -530.946,E2 -530.946} C_VEL
LIN {X 0,Y 608.47,Z 991.545,A -85,B 0,C 180,E1 -531.323,E2 -531.323} C_VEL
LIN {X 0,Y 608.478,Z 1001.441,A -85,B 0,C 180,E1 -531.783,E2 -531.783} C_VEL
LIN {X 0,Y 608.461,Z 1009.893,A -85,B 0,C 180,E1 -532.284,E2 -532.284} C_VEL
LIN {X 0,Y 608.458,Z 1017.859,A -85,B 0,C 180,E1 -532.868,E2 -532.868} C_VEL
LIN {X 0,Y 608.467,Z 1024.906,A -85,B 0,C 180,E1 -533.496,E2 -533.496} C_VEL
LIN {X 0,Y 608.458,Z 1031.401,A -85,B 0,C 180,E1 -534.2,E2 -534.2} C_VEL
LIN {X 0,Y 608.436,Z 1037.645,A -85,B 0,C 180,E1 -535.03,E2 -535.03} C_VEL
LIN {X 0,Y 608.432,Z 1043.428,A -85,B 0,C 180,E1 -536.026,E2 -536.026} C_VEL
LIN {X 0,Y 608.447,Z 1047.632,A -85,B 0,C 180,E1 -537.021,E2 -537.021} C_VEL
LIN {X 0,Y 608.443,Z 1050.571,A -85,B 0,C 180,E1 -538.014,E2 -538.014} C_VEL
LIN {X 0,Y 608.445,Z 1051.871,A -85,B 0,C 180,E1 -538.677,E2 -538.677} C_VEL
LIN {X 0,Y 608.434,Z 1052.693,A -85,B 0,C 180,E1 -539.338,E2 -539.338} C_VEL
LIN {X 0,Y 608.432,Z 1052.995,A -85,B 0,C 180,E1 -540,E2 -540} C_VEL
LIN {X 0,Y 608.435,Z 1052.735,A -85,B 0,C 180,E1 -540.662,E2 -540.662} C_VEL
LIN {X 0,Y 608.446,Z 1051.998,A -85,B 0,C 180,E1 -541.324,E2 -541.324} C_VEL
LIN {X 0,Y 608.444,Z 1050.787,A -85,B 0,C 180,E1 -541.986,E2 -541.986} C_VEL
LIN {X 0,Y 608.445,Z 1047.941,A -85,B 0,C 180,E1 -542.98,E2 -542.98} C_VEL
LIN {X 0,Y 608.444,Z 1045.352,A -85,B 0,C 180,E1 -543.643,E2 -543.643} C_VEL
LIN {X 0,Y 608.445,Z 1040.244,A -85,B 0,C 180,E1 -544.638,E2 -544.638} C_VEL
LIN {X 0,Y 608.461,Z 1034.747,A -85,B 0,C 180,E1 -545.468,E2 -545.468} C_VEL
LIN {X 0,Y 608.454,Z 1027.151,A -85,B 0,C 180,E1 -546.374,E2 -546.374} C_VEL
LIN {X 0,Y 608.462,Z 1018.945,A -85,B 0,C 180,E1 -547.133,E2 -547.133} C_VEL
LIN {X 0,Y 608.459,Z 1011.197,A -85,B 0,C 180,E1 -547.717,E2 -547.717} C_VEL
LIN {X 0,Y 608.478,Z 1003.03,A -85,B 0,C 180,E1 -548.218,E2 -548.218} C_VEL
LIN {X 0,Y 608.503,Z 999.979,A -85,B 0,C 180,E1 -548.386,E2 -548.386} C_VEL
LIN {X 0,Y 607.89,Z 994.713,A -85,B 0,C 180,E1 -548.639,E2 -548.639} C_VEL
LIN {X 0,Y 604.898,Z 986.088,A -85,B 0,C 180,E1 -549.016,E2 -549.016} C_VEL
LIN {X 0,Y 602.069,Z 977.176,A -85,B 0,C 180,E1 -549.32,E2 -549.32} C_VEL
LIN {X 0,Y 601.466,Z 971.475,A -85,B 0,C 180,E1 -549.443,E2 -549.443} C_VEL
LIN {X 0,Y 601.495,Z 945.566,A -85,B 0,C 180,E1 -549.776,E2 -549.776} C_VEL
LIN {X 0,Y 601.378,Z 894.674,A -85,B 0,C 180,E1 -550.383,E2 -550.383} C_VEL
LIN {X 0,Y 601.402,Z 881.043,A -85,B 0,C 180,E1 -553.173,E2 -553.173} C_VEL
LIN {X 0,Y 601.389,Z 869.344,A -85,B 0,C 180,E1 -555.592,E2 -555.592} C_VEL
LIN {X 0,Y 601.372,Z 860.384,A -85,B 0,C 180,E1 -557.47,E2 -557.47} C_VEL
LIN {X 0,Y 601.365,Z 860.382,A -85,B 0,C 180,E1 -559.811,E2 -559.811} C_VEL
LIN {X 0,Y 601.358,Z 860.383,A -85,B 0,C 180,E1 -561.962,E2 -561.962} C_VEL
LIN {X 0,Y 601.379,Z 860.384,A -85,B 0,C 180,E1 -564.88,E2 -564.88} C_VEL
LIN {X 0,Y 601.405,Z 860.388,A -85,B 0,C 180,E1 -567.36,E2 -567.36} C_VEL
LIN {X 0,Y 601.371,Z 860.382,A -85,B 0,C 180,E1 -570.168,E2 -570.168} C_VEL
LIN {X 0,Y 601.375,Z 860.38,A -85,B 0,C 180,E1 -572.708,E2 -572.708} C_VEL
LIN {X 0,Y 601.362,Z 860.384,A -85,B 0,C 180,E1 -575.107,E2 -575.107} C_VEL
LIN {X 0,Y 601.395,Z 860.382,A -85,B 0,C 180,E1 -577.423,E2 -577.423} C_VEL
LIN {X 0,Y 601.377,Z 860.391,A -85,B 0,C 180,E1 -579.998,E2 -579.998} C_VEL
LIN {X 0,Y 601.35,Z 860.385,A -85,B 0,C 180,E1 -582.676,E2 -582.676} C_VEL
LIN {X 0,Y 601.401,Z 860.381,A -85,B 0,C 180,E1 -584.533,E2 -584.533} C_VEL
LIN {X 0,Y 601.405,Z 860.384,A -85,B 0,C 180,E1 -586.43,E2 -586.43} C_VEL
LIN {X 0,Y 601.349,Z 860.384,A -85,B 0,C 180,E1 -589.12,E2 -589.12} C_VEL
LIN {X 0,Y 601.363,Z 860.382,A -85,B 0,C 180,E1 -591.538,E2 -591.538} C_VEL
LIN {X 0,Y 601.376,Z 860.386,A -85,B 0,C 180,E1 -594.245,E2 -594.245} C_VEL
LIN {X 0,Y 601.408,Z 860.388,A -85,B 0,C 180,E1 -596.685,E2 -596.685} C_VEL
LIN {X 0,Y 601.389,Z 860.385,A -85,B 0,C 180,E1 -599.056,E2 -599.056} C_VEL
LIN {X 0,Y 601.386,Z 860.382,A -85,B 0,C 180,E1 -601.371,E2 -601.371} C_VEL
LIN {X 0,Y 601.37,Z 860.382,A -85,B 0,C 180,E1 -603.635,E2 -603.635} C_VEL
LIN {X 0,Y 601.357,Z 860.383,A -85,B 0,C 180,E1 -605.855,E2 -605.855} C_VEL
LIN {X 0,Y 601.361,Z 860.382,A -85,B 0,C 180,E1 -608.039,E2 -608.039} C_VEL
LIN {X 0,Y 601.363,Z 860.382,A -85,B 0,C 180,E1 -610.189,E2 -610.189} C_VEL
LIN {X 0,Y 601.352,Z 860.383,A -85,B 0,C 180,E1 -612.31,E2 -612.31} C_VEL
LIN {X 0,Y 601.363,Z 860.382,A -85,B 0,C 180,E1 -614.407,E2 -614.407} C_VEL
LIN {X 0,Y 601.396,Z 860.382,A -85,B 0,C 180,E1 -617.171,E2 -617.171} C_VEL
LIN {X 0,Y 601.385,Z 860.387,A -85,B 0,C 180,E1 -619.904,E2 -619.904} C_VEL
LIN {X 0,Y 601.359,Z 860.383,A -85,B 0,C 180,E1 -622.614,E2 -622.614} C_VEL
LIN {X 0,Y 601.38,Z 860.381,A -85,B 0,C 180,E1 -625.308,E2 -625.308} C_VEL
LIN {X 0,Y 601.433,Z 860.384,A -85,B 0,C 180,E1 -627.991,E2 -627.991} C_VEL
LIN {X 0,Y 601.366,Z 860.385,A -85,B 0,C 180,E1 -630.67,E2 -630.67} C_VEL
LIN {X 0,Y 601.406,Z 860.381,A -85,B 0,C 180,E1 -632.679,E2 -632.679} C_VEL
LIN {X 0,Y 601.37,Z 860.381,A -85,B 0,C 180,E1 -635.365,E2 -635.365} C_VEL
LIN {X 0,Y 601.389,Z 860.382,A -85,B 0,C 180,E1 -638.062,E2 -638.062} C_VEL
LIN {X 0,Y 601.375,Z 860.385,A -85,B 0,C 180,E1 -640.984,E2 -640.984} C_VEL
LIN {X 0,Y 601.365,Z 860.382,A -85,B 0,C 180,E1 -643.517,E2 -643.517} C_VEL
LIN {X 0,Y 601.402,Z 860.379,A -85,B 0,C 180,E1 -646.288,E2 -646.288} C_VEL
LIN {X 0,Y 601.402,Z 860.387,A -85,B 0,C 180,E1 -649.1,E2 -649.1} C_VEL
LIN {X 0,Y 601.384,Z 860.388,A -85,B 0,C 180,E1 -651.24,E2 -651.24} C_VEL
LIN {X 0,Y 601.37,Z 860.381,A -85,B 0,C 180,E1 -654.277,E2 -654.277} C_VEL
LIN {X 0,Y 601.422,Z 860.382,A -85,B 0,C 180,E1 -657.113,E2 -657.113} C_VEL
LIN {X 0,Y 601.38,Z 860.391,A -85,B 0,C 180,E1 -659.395,E2 -659.395} C_VEL
LIN {X 0,Y 601.381,Z 860.388,A -85,B 0,C 180,E1 -661.728,E2 -661.728} C_VEL
LIN {X 0,Y 601.4,Z 860.381,A -85,B 0,C 180,E1 -664.121,E2 -664.121} C_VEL
LIN {X 0,Y 601.365,Z 860.382,A -85,B 0,C 180,E1 -666.586,E2 -666.586} C_VEL
LIN {X 0,Y 601.398,Z 860.382,A -85,B 0,C 180,E1 -669.53,E2 -669.53} C_VEL
LIN {X 0,Y 601.411,Z 860.383,A -85,B 0,C 180,E1 -671.767,E2 -671.767} C_VEL
LIN {X 0,Y 601.375,Z 860.384,A -85,B 0,C 180,E1 -674.53,E2 -674.53} C_VEL
LIN {X 0,Y 601.406,Z 860.384,A -85,B 0,C 180,E1 -676.43,E2 -676.43} C_VEL
LIN {X 0,Y 601.35,Z 860.384,A -85,B 0,C 180,E1 -679.12,E2 -679.12} C_VEL
LIN {X 0,Y 601.362,Z 860.382,A -85,B 0,C 180,E1 -681.538,E2 -681.538} C_VEL
LIN {X 0,Y 601.376,Z 860.386,A -85,B 0,C 180,E1 -684.244,E2 -684.244} C_VEL
LIN {X 0,Y 601.408,Z 860.388,A -85,B 0,C 180,E1 -686.685,E2 -686.685} C_VEL
LIN {X 0,Y 601.387,Z 860.385,A -85,B 0,C 180,E1 -689.056,E2 -689.056} C_VEL
LIN {X 0,Y 601.384,Z 860.382,A -85,B 0,C 180,E1 -691.37,E2 -691.37} C_VEL
LIN {X 0,Y 601.37,Z 860.382,A -85,B 0,C 180,E1 -693.634,E2 -693.634} C_VEL
LIN {X 0,Y 601.356,Z 860.383,A -85,B 0,C 180,E1 -695.855,E2 -695.855} C_VEL
LIN {X 0,Y 601.36,Z 860.382,A -85,B 0,C 180,E1 -698.038,E2 -698.038} C_VEL
LIN {X 0,Y 601.36,Z 860.382,A -85,B 0,C 180,E1 -700.189,E2 -700.189} C_VEL
LIN {X 0,Y 601.35,Z 860.383,A -85,B 0,C 180,E1 -702.31,E2 -702.31} C_VEL
LIN {X 0,Y 601.361,Z 860.382,A -85,B 0,C 180,E1 -704.407,E2 -704.407} C_VEL
LIN {X 0,Y 601.395,Z 860.382,A -85,B 0,C 180,E1 -707.171,E2 -707.171} C_VEL
LIN {X 0,Y 601.383,Z 860.387,A -85,B 0,C 180,E1 -709.904,E2 -709.904} C_VEL
LIN {X 0,Y 601.357,Z 860.383,A -85,B 0,C 180,E1 -712.614,E2 -712.614} C_VEL
LIN {X 0,Y 601.379,Z 860.382,A -85,B 0,C 180,E1 -715.307,E2 -715.307} C_VEL
LIN {X 0,Y 601.433,Z 860.384,A -85,B 0,C 180,E1 -717.991,E2 -717.991} C_VEL
LIN {X 0,Y 601.364,Z 860.384,A -85,B 0,C 180,E1 -720.669,E2 -720.669} C_VEL
LIN {X 0,Y 601.403,Z 860.381,A -85,B 0,C 180,E1 -722.679,E2 -722.679} C_VEL
LIN {X 0,Y 601.368,Z 860.381,A -85,B 0,C 180,E1 -725.364,E2 -725.364} C_VEL
LIN {X 0,Y 601.387,Z 860.383,A -85,B 0,C 180,E1 -728.061,E2 -728.061} C_VEL
LIN {X 0,Y 601.372,Z 860.385,A -85,B 0,C 180,E1 -730.984,E2 -730.984} C_VEL
LIN {X 0,Y 601.362,Z 860.382,A -85,B 0,C 180,E1 -733.517,E2 -733.517} C_VEL
LIN {X 0,Y 601.401,Z 860.379,A -85,B 0,C 180,E1 -736.288,E2 -736.288} C_VEL
LIN {X 0,Y 601.399,Z 860.387,A -85,B 0,C 180,E1 -739.099,E2 -739.099} C_VEL
LIN {X 0,Y 601.382,Z 860.388,A -85,B 0,C 180,E1 -741.24,E2 -741.24} C_VEL
LIN {X 0,Y 601.367,Z 860.381,A -85,B 0,C 180,E1 -744.277,E2 -744.277} C_VEL
LIN {X 0,Y 601.42,Z 860.382,A -85,B 0,C 180,E1 -747.112,E2 -747.112} C_VEL
LIN {X 0,Y 601.377,Z 860.392,A -85,B 0,C 180,E1 -749.395,E2 -749.395} C_VEL
LIN {X 0,Y 601.377,Z 860.388,A -85,B 0,C 180,E1 -751.728,E2 -751.728} C_VEL
LIN {X 0,Y 601.397,Z 860.381,A -85,B 0,C 180,E1 -754.12,E2 -754.12} C_VEL
LIN {X 0,Y 601.362,Z 860.382,A -85,B 0,C 180,E1 -756.586,E2 -756.586} C_VEL
LIN {X 0,Y 601.396,Z 860.383,A -85,B 0,C 180,E1 -759.53,E2 -759.53} C_VEL
LIN {X 0,Y 601.408,Z 860.384,A -85,B 0,C 180,E1 -761.766,E2 -761.766} C_VEL
LIN {X 0,Y 601.399,Z 860.381,A -85,B 0,C 180,E1 -764.532,E2 -764.532} C_VEL
LIN {X 0,Y 601.341,Z 860.385,A -85,B 0,C 180,E1 -767.323,E2 -767.323} C_VEL
LIN {X 0,Y 601.349,Z 860.383,A -85,B 0,C 180,E1 -769.434,E2 -769.434} C_VEL
LIN {X 0,Y 601.348,Z 860.385,A -85,B 0,C 180,E1 -771.726,E2 -771.726} C_VEL
LIN {X 0,Y 601.373,Z 860.387,A -85,B 0,C 180,E1 -774.244,E2 -774.244} C_VEL
LIN {X 0,Y 601.404,Z 860.388,A -85,B 0,C 180,E1 -776.685,E2 -776.685} C_VEL
LIN {X 0,Y 601.384,Z 860.385,A -85,B 0,C 180,E1 -779.056,E2 -779.056} C_VEL
LIN {X 0,Y 601.381,Z 860.382,A -85,B 0,C 180,E1 -781.37,E2 -781.37} C_VEL
LIN {X 0,Y 601.367,Z 860.383,A -85,B 0,C 180,E1 -783.634,E2 -783.634} C_VEL
LIN {X 0,Y 601.374,Z 860.381,A -85,B 0,C 180,E1 -785.856,E2 -785.856} C_VEL
LIN {X 0,Y 601.38,Z 860.525,A -85,B 0,C 180,E1 -788.355,E2 -788.355} C_VEL
LIN {X 0,Y 601.514,Z 868.62,A -85,B 0,C 180,E1 -789.66,E2 -789.66} C_VEL
LIN {X 0,Y 601.499,Z 884.252,A -85,B 0,C 180,E1 -792.139,E2 -792.139} C_VEL
LIN {X 0,Y 601.423,Z 901.001,A -85,B 0,C 180,E1 -794.756,E2 -794.756} C_VEL
LIN {X 0,Y 601.393,Z 919.983,A -85,B 0,C 180,E1 -797.686,E2 -797.686} C_VEL
LIN {X 0,Y 601.408,Z 932.684,A -85,B 0,C 180,E1 -799.628,E2 -799.628} C_VEL
LIN {X 0,Y 601.486,Z 1010.433,A -85,B 0,C 180,E1 -800.585,E2 -800.585} C_VEL
LIN {X 0,Y 601.485,Z 1020.898,A -85,B 0,C 180,E1 -800.818,E2 -800.818} C_VEL
LIN {X 0,Y 601.446,Z 1031.613,A -85,B 0,C 180,E1 -801.178,E2 -801.178} C_VEL
LIN {X 0,Y 601.448,Z 1042.231,A -85,B 0,C 180,E1 -801.686,E2 -801.686} C_VEL
LIN {X 0,Y 601.402,Z 1050.54,A -85,B 0,C 180,E1 -802.192,E2 -802.192} C_VEL
LIN {X 0,Y 601.409,Z 1058.399,A -85,B 0,C 180,E1 -802.783,E2 -802.783} C_VEL
LIN {X 0,Y 601.412,Z 1065.596,A -85,B 0,C 180,E1 -803.443,E2 -803.443} C_VEL
LIN {X 0,Y 601.391,Z 1073.19,A -85,B 0,C 180,E1 -804.299,E2 -804.299} C_VEL
LIN {X 0,Y 601.38,Z 1079.026,A -85,B 0,C 180,E1 -805.14,E2 -805.14} C_VEL
LIN {X 0,Y 601.343,Z 1083.63,A -85,B 0,C 180,E1 -805.979,E2 -805.979} C_VEL
LIN {X 0,Y 601.344,Z 1086.621,A -85,B 0,C 180,E1 -806.65,E2 -806.65} C_VEL
LIN {X 0,Y 601.326,Z 1088.931,A -85,B 0,C 180,E1 -807.32,E2 -807.32} C_VEL
LIN {X 0,Y 601.342,Z 1090.678,A -85,B 0,C 180,E1 -807.991,E2 -807.991} C_VEL
LIN {X 0,Y 601.345,Z 1091.934,A -85,B 0,C 180,E1 -808.661,E2 -808.661} C_VEL
LIN {X 0,Y 601.335,Z 1092.714,A -85,B 0,C 180,E1 -809.33,E2 -809.33} C_VEL
LIN {X 0,Y 601.332,Z 1093,A -85,B 0,C 180,E1 -810,E2 -810} C_VEL
LIN {X 0,Y 601.335,Z 1092.714,A -85,B 0,C 180,E1 -810.67,E2 -810.67} C_VEL
LIN {X 0,Y 601.345,Z 1091.934,A -85,B 0,C 180,E1 -811.339,E2 -811.339} C_VEL
LIN {X 0,Y 601.342,Z 1090.679,A -85,B 0,C 180,E1 -812.009,E2 -812.009} C_VEL
LIN {X 0,Y 601.343,Z 1087.786,A -85,B 0,C 180,E1 -813.015,E2 -813.015} C_VEL
LIN {X 0,Y 601.364,Z 1085.147,A -85,B 0,C 180,E1 -813.685,E2 -813.685} C_VEL
LIN {X 0,Y 601.366,Z 1079.985,A -85,B 0,C 180,E1 -814.692,E2 -814.692} C_VEL
LIN {X 0,Y 601.383,Z 1074.43,A -85,B 0,C 180,E1 -815.533,E2 -815.533} C_VEL
LIN {X 0,Y 601.393,Z 1067.151,A -85,B 0,C 180,E1 -816.403,E2 -816.403} C_VEL
LIN {X 0,Y 601.413,Z 1059.417,A -85,B 0,C 180,E1 -817.132,E2 -817.132} C_VEL
LIN {X 0,Y 601.424,Z 1051.762,A -85,B 0,C 180,E1 -817.723,E2 -817.723} C_VEL
LIN {X 0,Y 601.454,Z 1043.722,A -85,B 0,C 180,E1 -818.23,E2 -818.23} C_VEL
LIN {X 0,Y 601.453,Z 1035.392,A -85,B 0,C 180,E1 -818.653,E2 -818.653} C_VEL
LIN {X 0,Y 601.446,Z 1026.891,A -85,B 0,C 180,E1 -818.991,E2 -818.991} C_VEL
LIN {X 0,Y 601.468,Z 1016.757,A -85,B 0,C 180,E1 -819.288,E2 -819.288} C_VEL
LIN {X 0,Y 601.501,Z 1005.066,A -85,B 0,C 180,E1 -819.499,E2 -819.499} C_VEL
LIN {X 0,Y 601.408,Z 932.686,A -85,B 0,C 180,E1 -820.372,E2 -820.372} C_VEL
LIN {X 0,Y 601.433,Z 914.402,A -85,B 0,C 180,E1 -823.171,E2 -823.171} C_VEL
LIN {X 0,Y 601.482,Z 896.536,A -85,B 0,C 180,E1 -825.937,E2 -825.937} C_VEL
LIN {X 0,Y 601.511,Z 879.452,A -85,B 0,C 180,E1 -828.618,E2 -828.618} C_VEL
LIN {X 0,Y 601.534,Z 861.922,A -85,B 0,C 180,E1 -831.414,E2 -831.414} C_VEL
LIN {X 0,Y 601.375,Z 860.384,A -85,B 0,C 180,E1 -831.69,E2 -831.69} C_VEL
LIN {X 0,Y 601.367,Z 860.383,A -85,B 0,C 180,E1 -834.278,E2 -834.278} C_VEL
LIN {X 0,Y 601.394,Z 860.385,A -85,B 0,C 180,E1 -837.359,E2 -837.359} C_VEL
LIN {X 0,Y 601.366,Z 860.382,A -85,B 0,C 180,E1 -840.167,E2 -840.167} C_VEL
LIN {X 0,Y 601.375,Z 860.382,A -85,B 0,C 180,E1 -842.709,E2 -842.709} C_VEL
LIN {X 0,Y 601.361,Z 860.387,A -85,B 0,C 180,E1 -845.107,E2 -845.107} C_VEL
LIN {X 0,Y 601.391,Z 860.388,A -85,B 0,C 180,E1 -847.422,E2 -847.422} C_VEL
LIN {X 0,Y 601.374,Z 860.386,A -85,B 0,C 180,E1 -849.998,E2 -849.998} C_VEL
LIN {X 0,Y 601.343,Z 860.385,A -85,B 0,C 180,E1 -852.584,E2 -852.584} C_VEL
LIN {X 0,Y 601.363,Z 860.383,A -85,B 0,C 180,E1 -854.529,E2 -854.529} C_VEL
LIN {X 0,Y 601.399,Z 860.381,A -85,B 0,C 180,E1 -856.43,E2 -856.43} C_VEL
LIN {X 0,Y 601.349,Z 860.383,A -85,B 0,C 180,E1 -859.12,E2 -859.12} C_VEL
LIN {X 0,Y 601.357,Z 860.386,A -85,B 0,C 180,E1 -861.727,E2 -861.727} C_VEL
LIN {X 0,Y 601.374,Z 860.391,A -85,B 0,C 180,E1 -864.245,E2 -864.245} C_VEL
LIN {X 0,Y 601.402,Z 860.384,A -85,B 0,C 180,E1 -866.685,E2 -866.685} C_VEL
LIN {X 0,Y 601.379,Z 860.383,A -85,B 0,C 180,E1 -869.056,E2 -869.056} C_VEL
LIN {X 0,Y 601.374,Z 860.381,A -85,B 0,C 180,E1 -871.37,E2 -871.37} C_VEL
LIN {X 0,Y 601.36,Z 860.382,A -85,B 0,C 180,E1 -873.634,E2 -873.634} C_VEL
LIN {X 0,Y 601.372,Z 860.381,A -85,B 0,C 180,E1 -875.856,E2 -875.856} C_VEL
LIN {X 0,Y 601.378,Z 860.388,A -85,B 0,C 180,E1 -878.76,E2 -878.76} C_VEL
LIN {X 0,Y 601.368,Z 860.385,A -85,B 0,C 180,E1 -881.607,E2 -881.607} C_VEL
LIN {X 0,Y 601.388,Z 860.562,A -85,B 0,C 180,E1 -882.663,E2 -882.663} C_VEL
LIN {X 0,Y 601.396,Z 873.926,A -85,B 0,C 180,E1 -885.449,E2 -885.449} C_VEL
LIN {X 0,Y 601.376,Z 887.291,A -85,B 0,C 180,E1 -888.199,E2 -888.199} C_VEL
LIN {X 0,Y 601.37,Z 894.6,A -85,B 0,C 180,E1 -889.692,E2 -889.692} C_VEL
LIN {X 0,Y 601.568,Z 905.843,A -85,B 0,C 180,E1 -889.844,E2 -889.844} C_VEL
LIN {X 0,Y 601.472,Z 970.303,A -85,B 0,C 180,E1 -890.628,E2 -890.628} C_VEL
LIN {X 0,Y 601.46,Z 979.985,A -85,B 0,C 180,E1 -890.839,E2 -890.839} C_VEL
LIN {X 0,Y 601.445,Z 991.558,A -85,B 0,C 180,E1 -891.22,E2 -891.22} C_VEL
LIN {X 0,Y 601.447,Z 1001.459,A -85,B 0,C 180,E1 -891.686,E2 -891.686} C_VEL
LIN {X 0,Y 601.407,Z 1009.909,A -85,B 0,C 180,E1 -892.193,E2 -892.193} C_VEL
LIN {X 0,Y 601.409,Z 1017.87,A -85,B 0,C 180,E1 -892.784,E2 -892.784} C_VEL
LIN {X 0,Y 601.412,Z 1025.157,A -85,B 0,C 180,E1 -893.444,E2 -893.444} C_VEL
LIN {X 0,Y 601.386,Z 1031.411,A -85,B 0,C 180,E1 -894.131,E2 -894.131} C_VEL
LIN {X 0,Y 601.347,Z 1037.653,A -85,B 0,C 180,E1 -894.972,E2 -894.972} C_VEL
LIN {X 0,Y 601.344,Z 1043.435,A -85,B 0,C 180,E1 -895.979,E2 -895.979} C_VEL
LIN {X 0,Y 601.345,Z 1047.638,A -85,B 0,C 180,E1 -896.986,E2 -896.986} C_VEL
LIN {X 0,Y 601.342,Z 1050.576,A -85,B 0,C 180,E1 -897.991,E2 -897.991} C_VEL
LIN {X 0,Y 601.345,Z 1051.877,A -85,B 0,C 180,E1 -898.661,E2 -898.661} C_VEL
LIN {X 0,Y 601.335,Z 1052.697,A -85,B 0,C 180,E1 -899.331,E2 -899.331} C_VEL
LIN {X 0,Y 601.333,Z 1052.996,A -85,B 0,C 180,E1 -900,E2 -900} C_VEL
LIN {X 0,Y 601.336,Z 1052.738,A -85,B 0,C 180,E1 -900.67,E2 -900.67} C_VEL
LIN {X 0,Y 601.346,Z 1052.002,A -85,B 0,C 180,E1 -901.34,E2 -901.34} C_VEL
LIN {X 0,Y 601.343,Z 1050.79,A -85,B 0,C 180,E1 -902.01,E2 -902.01} C_VEL
LIN {X 0,Y 601.344,Z 1047.943,A -85,B 0,C 180,E1 -903.015,E2 -903.015} C_VEL
LIN {X 0,Y 601.363,Z 1045.355,A -85,B 0,C 180,E1 -903.686,E2 -903.686} C_VEL
LIN {X 0,Y 601.362,Z 1040.245,A -85,B 0,C 180,E1 -904.693,E2 -904.693} C_VEL
LIN {X 0,Y 601.384,Z 1034.748,A -85,B 0,C 180,E1 -905.533,E2 -905.533} C_VEL
LIN {X 0,Y 601.394,Z 1026.592,A -85,B 0,C 180,E1 -906.504,E2 -906.504} C_VEL
LIN {X 0,Y 601.412,Z 1018.943,A -85,B 0,C 180,E1 -907.217,E2 -907.217} C_VEL
LIN {X 0,Y 601.402,Z 1011.197,A -85,B 0,C 180,E1 -907.808,E2 -907.808} C_VEL
LIN {X 0,Y 601.448,Z 1003.03,A -85,B 0,C 180,E1 -908.315,E2 -908.315} C_VEL
LIN {X 0,Y 601.432,Z 992.651,A -85,B 0,C 180,E1 -908.823,E2 -908.823} C_VEL
LIN {X 0,Y 601.449,Z 980.995,A -85,B 0,C 180,E1 -909.225,E2 -909.225} C_VEL
LIN {X 0,Y 601.466,Z 971.475,A -85,B 0,C 180,E1 -909.443,E2 -909.443} C_VEL
LIN {X 0,Y 600.888,Z 965.689,A -85,B 0,C 180,E1 -909.546,E2 -909.546} C_VEL
LIN {X 0,Y 595.142,Z 946.982,A -85,B 0,C 180,E1 -909.865,E2 -909.865} C_VEL
LIN {X 0,Y 594.51,Z 941.164,A -85,B 0,C 180,E1 -909.944,E2 -909.944} C_VEL
LIN {X 0,Y 594.379,Z 895.429,A -85,B 0,C 180,E1 -910.496,E2 -910.496} C_VEL
LIN {X 0,Y 594.293,Z 894.619,A -85,B 0,C 180,E1 -910.519,E2 -910.519} C_VEL
LIN {X 0,Y 594.361,Z 881.04,A -85,B 0,C 180,E1 -913.331,E2 -913.331} C_VEL
LIN {X 0,Y 594.354,Z 867.67,A -85,B 0,C 180,E1 -916.134,E2 -916.134} C_VEL
LIN {X 0,Y 594.329,Z 861.261,A -85,B 0,C 180,E1 -917.506,E2 -917.506} C_VEL
LIN {X 0,Y 594.34,Z 861.257,A -85,B 0,C 180,E1 -920.055,E2 -920.055} C_VEL
LIN {X 0,Y 594.323,Z 861.266,A -85,B 0,C 180,E1 -922.969,E2 -922.969} C_VEL
LIN {X 0,Y 594.341,Z 861.267,A -85,B 0,C 180,E1 -925.195,E2 -925.195} C_VEL
LIN {X 0,Y 594.345,Z 861.265,A -85,B 0,C 180,E1 -927.519,E2 -927.519} C_VEL
LIN {X 0,Y 594.345,Z 861.256,A -85,B 0,C 180,E1 -930.321,E2 -930.321} C_VEL
LIN {X 0,Y 594.335,Z 861.259,A -85,B 0,C 180,E1 -932.953,E2 -932.953} C_VEL
LIN {X 0,Y 594.316,Z 861.265,A -85,B 0,C 180,E1 -935.412,E2 -935.412} C_VEL
LIN {X 0,Y 594.344,Z 861.266,A -85,B 0,C 180,E1 -937.944,E2 -937.944} C_VEL
LIN {X 0,Y 594.325,Z 861.26,A -85,B 0,C 180,E1 -940.571,E2 -940.571} C_VEL
LIN {X 0,Y 594.313,Z 861.26,A -85,B 0,C 180,E1 -942.847,E2 -942.847} C_VEL
LIN {X 0,Y 594.316,Z 861.26,A -85,B 0,C 180,E1 -945.197,E2 -945.197} C_VEL
LIN {X 0,Y 594.364,Z 861.263,A -85,B 0,C 180,E1 -948.154,E2 -948.154} C_VEL
LIN {X 0,Y 594.322,Z 861.26,A -85,B 0,C 180,E1 -951.19,E2 -951.19} C_VEL
LIN {X 0,Y 594.334,Z 861.258,A -85,B 0,C 180,E1 -953.754,E2 -953.754} C_VEL
LIN {X 0,Y 594.359,Z 861.258,A -85,B 0,C 180,E1 -956.238,E2 -956.238} C_VEL
LIN {X 0,Y 594.345,Z 861.266,A -85,B 0,C 180,E1 -958.648,E2 -958.648} C_VEL
LIN {X 0,Y 594.341,Z 861.265,A -85,B 0,C 180,E1 -961.051,E2 -961.051} C_VEL
LIN {X 0,Y 594.355,Z 861.26,A -85,B 0,C 180,E1 -963.299,E2 -963.299} C_VEL
LIN {X 0,Y 594.321,Z 861.259,A -85,B 0,C 180,E1 -966.293,E2 -966.293} C_VEL
LIN {X 0,Y 594.396,Z 861.262,A -85,B 0,C 180,E1 -969.224,E2 -969.224} C_VEL
LIN {X 0,Y 594.314,Z 861.261,A -85,B 0,C 180,E1 -972.094,E2 -972.094} C_VEL
LIN {X 0,Y 594.323,Z 861.259,A -85,B 0,C 180,E1 -974.218,E2 -974.218} C_VEL
LIN {X 0,Y 594.336,Z 861.258,A -85,B 0,C 180,E1 -976.32,E2 -976.32} C_VEL
LIN {X 0,Y 594.336,Z 861.258,A -85,B 0,C 180,E1 -978.956,E2 -978.956} C_VEL
LIN {X 0,Y 594.35,Z 861.266,A -85,B 0,C 180,E1 -981.843,E2 -981.843} C_VEL
LIN {X 0,Y 594.343,Z 861.258,A -85,B 0,C 180,E1 -984.572,E2 -984.572} C_VEL
LIN {X 0,Y 594.363,Z 861.255,A -85,B 0,C 180,E1 -987.289,E2 -987.289} C_VEL
LIN {X 0,Y 594.413,Z 861.256,A -85,B 0,C 180,E1 -990,E2 -990} C_VEL
LIN {X 0,Y 594.372,Z 861.256,A -85,B 0,C 180,E1 -992.711,E2 -992.711} C_VEL
LIN {X 0,Y 594.34,Z 861.257,A -85,B 0,C 180,E1 -995.428,E2 -995.428} C_VEL
LIN {X 0,Y 594.346,Z 861.261,A -85,B 0,C 180,E1 -998.158,E2 -998.158} C_VEL
LIN {X 0,Y 594.336,Z 861.261,A -85,B 0,C 180,E1 -1001.044,E2 -1001.044} C_VEL
LIN {X 0,Y 594.335,Z 861.257,A -85,B 0,C 180,E1 -1003.68,E2 -1003.68} C_VEL
LIN {X 0,Y 594.355,Z 861.263,A -85,B 0,C 180,E1 -1006.705,E2 -1006.705} C_VEL
LIN {X 0,Y 594.349,Z 861.261,A -85,B 0,C 180,E1 -1009.335,E2 -1009.335} C_VEL
LIN {X 0,Y 594.336,Z 861.261,A -85,B 0,C 180,E1 -1011.505,E2 -1011.505} C_VEL
LIN {X 0,Y 594.343,Z 861.257,A -85,B 0,C 180,E1 -1014.448,E2 -1014.448} C_VEL
LIN {X 0,Y 594.345,Z 861.266,A -85,B 0,C 180,E1 -1017.463,E2 -1017.463} C_VEL
LIN {X 0,Y 594.348,Z 861.256,A -85,B 0,C 180,E1 -1020.321,E2 -1020.321} C_VEL
LIN {X 0,Y 594.336,Z 861.259,A -85,B 0,C 180,E1 -1022.953,E2 -1022.953} C_VEL
LIN {X 0,Y 594.316,Z 861.266,A -85,B 0,C 180,E1 -1025.412,E2 -1025.412} C_VEL
LIN {X 0,Y 594.312,Z 861.27,A -85,B 0,C 180,E1 -1027.947,E2 -1027.947} C_VEL
LIN {X 0,Y 594.327,Z 861.26,A -85,B 0,C 180,E1 -1030.571,E2 -1030.571} C_VEL
LIN {X 0,Y 594.312,Z 861.261,A -85,B 0,C 180,E1 -1032.846,E2 -1032.846} C_VEL
LIN {X 0,Y 594.309,Z 861.26,A -85,B 0,C 180,E1 -1035.197,E2 -1035.197} C_VEL
LIN {X 0,Y 594.364,Z 861.263,A -85,B 0,C 180,E1 -1038.154,E2 -1038.154} C_VEL
LIN {X 0,Y 594.322,Z 861.259,A -85,B 0,C 180,E1 -1041.19,E2 -1041.19} C_VEL
LIN {X 0,Y 594.334,Z 861.258,A -85,B 0,C 180,E1 -1043.754,E2 -1043.754} C_VEL
LIN {X 0,Y 594.359,Z 861.259,A -85,B 0,C 180,E1 -1046.237,E2 -1046.237} C_VEL
LIN {X 0,Y 594.344,Z 861.266,A -85,B 0,C 180,E1 -1048.648,E2 -1048.648} C_VEL
LIN {X 0,Y 594.341,Z 861.264,A -85,B 0,C 180,E1 -1051.05,E2 -1051.05} C_VEL
LIN {X 0,Y 594.355,Z 861.26,A -85,B 0,C 180,E1 -1053.299,E2 -1053.299} C_VEL
LIN {X 0,Y 594.319,Z 861.26,A -85,B 0,C 180,E1 -1056.293,E2 -1056.293} C_VEL
LIN {X 0,Y 594.394,Z 861.262,A -85,B 0,C 180,E1 -1059.224,E2 -1059.224} C_VEL
LIN {X 0,Y 594.313,Z 861.261,A -85,B 0,C 180,E1 -1062.093,E2 -1062.093} C_VEL
LIN {X 0,Y 594.321,Z 861.259,A -85,B 0,C 180,E1 -1064.217,E2 -1064.217} C_VEL
LIN {X 0,Y 594.335,Z 861.26,A -85,B 0,C 180,E1 -1067.016,E2 -1067.016} C_VEL
LIN {X 0,Y 594.332,Z 861.267,A -85,B 0,C 180,E1 -1069.783,E2 -1069.783} C_VEL
LIN {X 0,Y 594.334,Z 861.258,A -85,B 0,C 180,E1 -1072.526,E2 -1072.526} C_VEL
LIN {X 0,Y 594.35,Z 861.257,A -85,B 0,C 180,E1 -1075.252,E2 -1075.252} C_VEL
LIN {X 0,Y 594.401,Z 861.26,A -85,B 0,C 180,E1 -1077.967,E2 -1077.967} C_VEL
LIN {X 0,Y 594.319,Z 861.262,A -85,B 0,C 180,E1 -1080.677,E2 -1080.677} C_VEL
LIN {X 0,Y 594.369,Z 861.257,A -85,B 0,C 180,E1 -1082.711,E2 -1082.711} C_VEL
LIN {X 0,Y 594.338,Z 861.257,A -85,B 0,C 180,E1 -1085.428,E2 -1085.428} C_VEL
LIN {X 0,Y 594.344,Z 861.262,A -85,B 0,C 180,E1 -1088.157,E2 -1088.157} C_VEL
LIN {X 0,Y 594.333,Z 861.261,A -85,B 0,C 180,E1 -1091.044,E2 -1091.044} C_VEL
LIN {X 0,Y 594.332,Z 861.258,A -85,B 0,C 180,E1 -1093.68,E2 -1093.68} C_VEL
LIN {X 0,Y 594.354,Z 861.264,A -85,B 0,C 180,E1 -1096.705,E2 -1096.705} C_VEL
LIN {X 0,Y 594.346,Z 861.261,A -85,B 0,C 180,E1 -1099.335,E2 -1099.335} C_VEL
LIN {X 0,Y 594.333,Z 861.261,A -85,B 0,C 180,E1 -1101.504,E2 -1101.504} C_VEL
LIN {X 0,Y 594.339,Z 861.257,A -85,B 0,C 180,E1 -1104.448,E2 -1104.448} C_VEL
LIN {X 0,Y 594.342,Z 861.266,A -85,B 0,C 180,E1 -1107.462,E2 -1107.462} C_VEL
LIN {X 0,Y 594.344,Z 861.256,A -85,B 0,C 180,E1 -1110.32,E2 -1110.32} C_VEL
LIN {X 0,Y 594.333,Z 861.259,A -85,B 0,C 180,E1 -1112.953,E2 -1112.953} C_VEL
LIN {X 0,Y 594.314,Z 861.266,A -85,B 0,C 180,E1 -1115.411,E2 -1115.411} C_VEL
LIN {X 0,Y 594.34,Z 861.266,A -85,B 0,C 180,E1 -1117.944,E2 -1117.944} C_VEL
LIN {X 0,Y 594.323,Z 861.26,A -85,B 0,C 180,E1 -1120.571,E2 -1120.571} C_VEL
LIN {X 0,Y 594.309,Z 861.261,A -85,B 0,C 180,E1 -1122.846,E2 -1122.846} C_VEL
LIN {X 0,Y 594.313,Z 861.26,A -85,B 0,C 180,E1 -1125.196,E2 -1125.196} C_VEL
LIN {X 0,Y 594.362,Z 861.264,A -85,B 0,C 180,E1 -1128.154,E2 -1128.154} C_VEL
LIN {X 0,Y 594.318,Z 861.26,A -85,B 0,C 180,E1 -1131.19,E2 -1131.19} C_VEL
LIN {X 0,Y 594.331,Z 861.258,A -85,B 0,C 180,E1 -1133.754,E2 -1133.754} C_VEL
LIN {X 0,Y 594.355,Z 861.259,A -85,B 0,C 180,E1 -1136.237,E2 -1136.237} C_VEL
LIN {X 0,Y 594.34,Z 861.267,A -85,B 0,C 180,E1 -1138.648,E2 -1138.648} C_VEL
LIN {X 0,Y 594.337,Z 861.264,A -85,B 0,C 180,E1 -1141.05,E2 -1141.05} C_VEL
LIN {X 0,Y 594.352,Z 861.261,A -85,B 0,C 180,E1 -1143.299,E2 -1143.299} C_VEL
LIN {X 0,Y 594.325,Z 861.26,A -85,B 0,C 180,E1 -1146.293,E2 -1146.293} C_VEL
LIN {X 0,Y 594.35,Z 861.363,A -85,B 0,C 180,E1 -1148.223,E2 -1148.223} C_VEL
LIN {X 0,Y 594.576,Z 867.504,A -85,B 0,C 180,E1 -1149.23,E2 -1149.23} C_VEL
LIN {X 0,Y 594.495,Z 883.136,A -85,B 0,C 180,E1 -1151.743,E2 -1151.743} C_VEL
LIN {X 0,Y 594.435,Z 899.884,A -85,B 0,C 180,E1 -1154.397,E2 -1154.397} C_VEL
LIN {X 0,Y 594.388,Z 917.75,A -85,B 0,C 180,E1 -1157.191,E2 -1157.191} C_VEL
LIN {X 0,Y 594.347,Z 932.754,A -85,B 0,C 180,E1 -1159.514,E2 -1159.514} C_VEL
LIN {X 0,Y 594.564,Z 962.115,A -85,B 0,C 180,E1 -1159.873,E2 -1159.873} C_VEL
LIN {X 0,Y 594.499,Z 1010.432,A -85,B 0,C 180,E1 -1160.473,E2 -1160.473} C_VEL
LIN {X 0,Y 594.483,Z 1020.898,A -85,B 0,C 180,E1 -1160.709,E2 -1160.709} C_VEL
LIN {X 0,Y 594.435,Z 1031.612,A -85,B 0,C 180,E1 -1161.073,E2 -1161.073} C_VEL
LIN {X 0,Y 594.428,Z 1042.233,A -85,B 0,C 180,E1 -1161.587,E2 -1161.587} C_VEL
LIN {X 0,Y 594.374,Z 1050.542,A -85,B 0,C 180,E1 -1162.099,E2 -1162.099} C_VEL
LIN {X 0,Y 594.351,Z 1058.399,A -85,B 0,C 180,E1 -1162.697,E2 -1162.697} C_VEL
LIN {X 0,Y 594.342,Z 1065.512,A -85,B 0,C 180,E1 -1163.356,E2 -1163.356} C_VEL
LIN {X 0,Y 594.318,Z 1073.189,A -85,B 0,C 180,E1 -1164.231,E2 -1164.231} C_VEL
LIN {X 0,Y 594.289,Z 1079.027,A -85,B 0,C 180,E1 -1165.081,E2 -1165.081} C_VEL
LIN {X 0,Y 594.26,Z 1083.63,A -85,B 0,C 180,E1 -1165.931,E2 -1165.931} C_VEL
LIN {X 0,Y 594.267,Z 1086.621,A -85,B 0,C 180,E1 -1166.61,E2 -1166.61} C_VEL
LIN {X 0,Y 594.228,Z 1088.931,A -85,B 0,C 180,E1 -1167.288,E2 -1167.288} C_VEL
LIN {X 0,Y 594.241,Z 1090.679,A -85,B 0,C 180,E1 -1167.967,E2 -1167.967} C_VEL
LIN {X 0,Y 594.245,Z 1091.934,A -85,B 0,C 180,E1 -1168.644,E2 -1168.644} C_VEL
LIN {X 0,Y 594.235,Z 1092.713,A -85,B 0,C 180,E1 -1169.322,E2 -1169.322} C_VEL
LIN {X 0,Y 594.233,Z 1093,A -85,B 0,C 180,E1 -1170,E2 -1170} C_VEL
LIN {X 0,Y 594.235,Z 1092.713,A -85,B 0,C 180,E1 -1170.678,E2 -1170.678} C_VEL
LIN {X 0,Y 594.245,Z 1091.935,A -85,B 0,C 180,E1 -1171.355,E2 -1171.355} C_VEL
LIN {X 0,Y 594.241,Z 1090.679,A -85,B 0,C 180,E1 -1172.033,E2 -1172.033} C_VEL
LIN {X 0,Y 594.246,Z 1087.787,A -85,B 0,C 180,E1 -1173.051,E2 -1173.051} C_VEL
LIN {X 0,Y 594.285,Z 1085.147,A -85,B 0,C 180,E1 -1173.729,E2 -1173.729} C_VEL
LIN {X 0,Y 594.276,Z 1079.986,A -85,B 0,C 180,E1 -1174.748,E2 -1174.748} C_VEL
LIN {X 0,Y 594.309,Z 1074.431,A -85,B 0,C 180,E1 -1175.599,E2 -1175.599} C_VEL
LIN {X 0,Y 594.344,Z 1067.15,A -85,B 0,C 180,E1 -1176.479,E2 -1176.479} C_VEL
LIN {X 0,Y 594.354,Z 1059.417,A -85,B 0,C 180,E1 -1177.217,E2 -1177.217} C_VEL
LIN {X 0,Y 594.358,Z 1051.764,A -85,B 0,C 180,E1 -1177.815,E2 -1177.815} C_VEL
LIN {X 0,Y 594.432,Z 1043.724,A -85,B 0,C 180,E1 -1178.327,E2 -1178.327} C_VEL
LIN {X 0,Y 594.425,Z 1035.394,A -85,B 0,C 180,E1 -1178.756,E2 -1178.756} C_VEL
LIN {X 0,Y 594.44,Z 1026.892,A -85,B 0,C 180,E1 -1179.098,E2 -1179.098} C_VEL
LIN {X 0,Y 594.476,Z 1016.758,A -85,B 0,C 180,E1 -1179.398,E2 -1179.398} C_VEL
LIN {X 0,Y 594.518,Z 1005.066,A -85,B 0,C 180,E1 -1179.612,E2 -1179.612} C_VEL
LIN {X 0,Y 594.43,Z 933.517,A -85,B 0,C 180,E1 -1180.473,E2 -1180.473} C_VEL
LIN {X 0,Y 594.351,Z 932.686,A -85,B 0,C 180,E1 -1180.496,E2 -1180.496} C_VEL
LIN {X 0,Y 594.378,Z 914.402,A -85,B 0,C 180,E1 -1183.331,E2 -1183.331} C_VEL
LIN {X 0,Y 594.463,Z 896.536,A -85,B 0,C 180,E1 -1186.13,E2 -1186.13} C_VEL
LIN {X 0,Y 594.539,Z 879.323,A -85,B 0,C 180,E1 -1188.866,E2 -1188.866} C_VEL
LIN {X 0,Y 594.555,Z 863.039,A -85,B 0,C 180,E1 -1191.496,E2 -1191.496} C_VEL
LIN {X 0,Y 594.333,Z 861.263,A -85,B 0,C 180,E1 -1191.823,E2 -1191.823} C_VEL
LIN {X 0,Y 594.337,Z 861.261,A -85,B 0,C 180,E1 -1194.448,E2 -1194.448} C_VEL
LIN {X 0,Y 594.335,Z 861.263,A -85,B 0,C 180,E1 -1197.463,E2 -1197.463} C_VEL
LIN {X 0,Y 594.341,Z 861.257,A -85,B 0,C 180,E1 -1200.321,E2 -1200.321} C_VEL
LIN {X 0,Y 594.336,Z 861.262,A -85,B 0,C 180,E1 -1202.953,E2 -1202.953} C_VEL
LIN {X 0,Y 594.313,Z 861.271,A -85,B 0,C 180,E1 -1205.412,E2 -1205.412} C_VEL
LIN {X 0,Y 594.304,Z 861.266,A -85,B 0,C 180,E1 -1207.947,E2 -1207.947} C_VEL
LIN {X 0,Y 594.302,Z 861.261,A -85,B 0,C 180,E1 -1210.572,E2 -1210.572} C_VEL
LIN {X 0,Y 594.304,Z 861.261,A -85,B 0,C 180,E1 -1212.846,E2 -1212.846} C_VEL
LIN {X 0,Y 594.305,Z 861.262,A -85,B 0,C 180,E1 -1215.197,E2 -1215.197} C_VEL
LIN {X 0,Y 594.363,Z 861.264,A -85,B 0,C 180,E1 -1218.154,E2 -1218.154} C_VEL
LIN {X 0,Y 594.318,Z 861.26,A -85,B 0,C 180,E1 -1221.19,E2 -1221.19} C_VEL
LIN {X 0,Y 594.33,Z 861.26,A -85,B 0,C 180,E1 -1223.754,E2 -1223.754} C_VEL
LIN {X 0,Y 594.354,Z 861.263,A -85,B 0,C 180,E1 -1226.237,E2 -1226.237} C_VEL
LIN {X 0,Y 594.338,Z 861.266,A -85,B 0,C 180,E1 -1228.648,E2 -1228.648} C_VEL
LIN {X 0,Y 594.335,Z 861.262,A -85,B 0,C 180,E1 -1231.051,E2 -1231.051} C_VEL
LIN {X 0,Y 594.345,Z 861.259,A -85,B 0,C 180,E1 -1233.299,E2 -1233.299} C_VEL
LIN {X 0,Y 594.323,Z 861.262,A -85,B 0,C 180,E1 -1236.293,E2 -1236.293} C_VEL
LIN {X 0,Y 594.382,Z 861.259,A -85,B 0,C 180,E1 -1239.224,E2 -1239.224} C_VEL
LIN {X 0,Y 594.355,Z 861.262,A -85,B 0,C 180,E1 -1241.382,E2 -1241.382} C_VEL
LIN {X 0,Y 594.361,Z 861.4,A -85,B 0,C 180,E1 -1242.629,E2 -1242.629} C_VEL
LIN {X 0,Y 594.347,Z 873.929,A -85,B 0,C 180,E1 -1245.272,E2 -1245.272} C_VEL
LIN {X 0,Y 594.321,Z 885.623,A -85,B 0,C 180,E1 -1247.711,E2 -1247.711} C_VEL
LIN {X 0,Y 594.291,Z 894.603,A -85,B 0,C 180,E1 -1249.567,E2 -1249.567} C_VEL
LIN {X 0,Y 594.578,Z 900.523,A -85,B 0,C 180,E1 -1249.659,E2 -1249.659} C_VEL
LIN {X 0,Y 594.491,Z 970.336,A -85,B 0,C 180,E1 -1250.517,E2 -1250.517} C_VEL
LIN {X 0,Y 594.46,Z 980.008,A -85,B 0,C 180,E1 -1250.731,E2 -1250.731} C_VEL
LIN {X 0,Y 594.42,Z 991.57,A -85,B 0,C 180,E1 -1251.116,E2 -1251.116} C_VEL
LIN {X 0,Y 594.427,Z 1001.477,A -85,B 0,C 180,E1 -1251.587,E2 -1251.587} C_VEL
LIN {X 0,Y 594.375,Z 1009.925,A -85,B 0,C 180,E1 -1252.1,E2 -1252.1} C_VEL
LIN {X 0,Y 594.351,Z 1017.88,A -85,B 0,C 180,E1 -1252.697,E2 -1252.697} C_VEL
LIN {X 0,Y 594.343,Z 1025.084,A -85,B 0,C 180,E1 -1253.357,E2 -1253.357} C_VEL
LIN {X 0,Y 594.318,Z 1032.834,A -85,B 0,C 180,E1 -1254.231,E2 -1254.231} C_VEL
LIN {X 0,Y 594.274,Z 1039.743,A -85,B 0,C 180,E1 -1255.252,E2 -1255.252} C_VEL
LIN {X 0,Y 594.286,Z 1044.959,A -85,B 0,C 180,E1 -1256.271,E2 -1256.271} C_VEL
LIN {X 0,Y 594.229,Z 1048.788,A -85,B 0,C 180,E1 -1257.289,E2 -1257.289} C_VEL
LIN {X 0,Y 594.241,Z 1050.581,A -85,B 0,C 180,E1 -1257.967,E2 -1257.967} C_VEL
LIN {X 0,Y 594.244,Z 1051.882,A -85,B 0,C 180,E1 -1258.645,E2 -1258.645} C_VEL
LIN {X 0,Y 594.235,Z 1052.7,A -85,B 0,C 180,E1 -1259.323,E2 -1259.323} C_VEL
LIN {X 0,Y 594.234,Z 1052.996,A -85,B 0,C 180,E1 -1260,E2 -1260} C_VEL
LIN {X 0,Y 594.236,Z 1052.741,A -85,B 0,C 180,E1 -1260.678,E2 -1260.678} C_VEL
LIN {X 0,Y 594.246,Z 1052.006,A -85,B 0,C 180,E1 -1261.356,E2 -1261.356} C_VEL
LIN {X 0,Y 594.242,Z 1050.792,A -85,B 0,C 180,E1 -1262.034,E2 -1262.034} C_VEL
LIN {X 0,Y 594.247,Z 1047.945,A -85,B 0,C 180,E1 -1263.051,E2 -1263.051} C_VEL
LIN {X 0,Y 594.285,Z 1045.358,A -85,B 0,C 180,E1 -1263.73,E2 -1263.73} C_VEL
LIN {X 0,Y 594.265,Z 1040.247,A -85,B 0,C 180,E1 -1264.749,E2 -1264.749} C_VEL
LIN {X 0,Y 594.309,Z 1034.749,A -85,B 0,C 180,E1 -1265.599,E2 -1265.599} C_VEL
LIN {X 0,Y 594.324,Z 1026.694,A -85,B 0,C 180,E1 -1266.57,E2 -1266.57} C_VEL
LIN {X 0,Y 594.353,Z 1018.94,A -85,B 0,C 180,E1 -1267.303,E2 -1267.303} C_VEL
LIN {X 0,Y 594.373,Z 1011.198,A -85,B 0,C 180,E1 -1267.901,E2 -1267.901} C_VEL
LIN {X 0,Y 594.427,Z 1003.03,A -85,B 0,C 180,E1 -1268.414,E2 -1268.414} C_VEL
LIN {X 0,Y 594.427,Z 992.636,A -85,B 0,C 180,E1 -1268.928,E2 -1268.928} C_VEL
LIN {X 0,Y 594.451,Z 980.976,A -85,B 0,C 180,E1 -1269.335,E2 -1269.335} C_VEL
LIN {X 0,Y 594.486,Z 970.548,A -85,B 0,C 180,E1 -1269.57,E2 -1269.57} C_VEL
LIN {X 0,Y 594.51,Z 941.164,A -85,B 0,C 180,E1 -1269.944,E2 -1269.944} C_VEL
LIN {X 0,Y 593.901,Z 935.348,A -85,B 0,C 180,E1 -1270.024,E2 -1270.024} C_VEL
LIN {X 0,Y 588.278,Z 916.608,A -85,B 0,C 180,E1 -1270.348,E2 -1270.348} C_VEL
LIN {X 0,Y 587.591,Z 910.793,A -85,B 0,C 180,E1 -1270.431,E2 -1270.431} C_VEL
LIN {X 0,Y 587.464,Z 896.388,A -85,B 0,C 180,E1 -1270.609,E2 -1270.609} C_VEL
LIN {X 0,Y 587.232,Z 894.638,A -85,B 0,C 180,E1 -1270.643,E2 -1270.643} C_VEL
LIN {X 0,Y 587.3,Z 881.038,A -85,B 0,C 180,E1 -1273.495,E2 -1273.495} C_VEL
LIN {X 0,Y 587.324,Z 867.667,A -85,B 0,C 180,E1 -1276.332,E2 -1276.332} C_VEL
LIN {X 0,Y 587.317,Z 862.135,A -85,B 0,C 180,E1 -1277.542,E2 -1277.542} C_VEL
LIN {X 0,Y 587.3,Z 862.134,A -85,B 0,C 180,E1 -1280.306,E2 -1280.306} C_VEL
LIN {X 0,Y 587.282,Z 862.146,A -85,B 0,C 180,E1 -1283.261,E2 -1283.261} C_VEL
LIN {X 0,Y 587.296,Z 862.135,A -85,B 0,C 180,E1 -1286.168,E2 -1286.168} C_VEL
LIN {X 0,Y 587.299,Z 862.139,A -85,B 0,C 180,E1 -1289.124,E2 -1289.124} C_VEL
LIN {X 0,Y 587.317,Z 862.138,A -85,B 0,C 180,E1 -1291.831,E2 -1291.831} C_VEL
LIN {X 0,Y 587.32,Z 862.133,A -85,B 0,C 180,E1 -1294.344,E2 -1294.344} C_VEL
LIN {X 0,Y 587.309,Z 862.14,A -85,B 0,C 180,E1 -1297.611,E2 -1297.611} C_VEL
LIN {X 0,Y 587.285,Z 862.141,A -85,B 0,C 180,E1 -1300.257,E2 -1300.257} C_VEL
LIN {X 0,Y 587.277,Z 862.136,A -85,B 0,C 180,E1 -1303.114,E2 -1303.114} C_VEL
LIN {X 0,Y 587.288,Z 862.144,A -85,B 0,C 180,E1 -1306.046,E2 -1306.046} C_VEL
LIN {X 0,Y 587.279,Z 862.138,A -85,B 0,C 180,E1 -1308.932,E2 -1308.932} C_VEL
LIN {X 0,Y 587.269,Z 862.138,A -85,B 0,C 180,E1 -1311.516,E2 -1311.516} C_VEL
LIN {X 0,Y 587.272,Z 862.141,A -85,B 0,C 180,E1 -1314.099,E2 -1314.099} C_VEL
LIN {X 0,Y 587.313,Z 862.143,A -85,B 0,C 180,E1 -1316.602,E2 -1316.602} C_VEL
LIN {X 0,Y 587.288,Z 862.136,A -85,B 0,C 180,E1 -1319.499,E2 -1319.499} C_VEL
LIN {X 0,Y 587.299,Z 862.136,A -85,B 0,C 180,E1 -1322.318,E2 -1322.318} C_VEL
LIN {X 0,Y 587.288,Z 862.143,A -85,B 0,C 180,E1 -1325.239,E2 -1325.239} C_VEL
LIN {X 0,Y 587.302,Z 862.139,A -85,B 0,C 180,E1 -1327.485,E2 -1327.485} C_VEL
LIN {X 0,Y 587.306,Z 862.137,A -85,B 0,C 180,E1 -1329.694,E2 -1329.694} C_VEL
LIN {X 0,Y 587.276,Z 862.139,A -85,B 0,C 180,E1 -1331.872,E2 -1331.872} C_VEL
LIN {X 0,Y 587.287,Z 862.137,A -85,B 0,C 180,E1 -1334.024,E2 -1334.024} C_VEL
LIN {X 0,Y 587.323,Z 862.133,A -85,B 0,C 180,E1 -1336.153,E2 -1336.153} C_VEL
LIN {X 0,Y 587.296,Z 862.135,A -85,B 0,C 180,E1 -1338.962,E2 -1338.962} C_VEL
LIN {X 0,Y 587.316,Z 862.143,A -85,B 0,C 180,E1 -1341.744,E2 -1341.744} C_VEL
LIN {X 0,Y 587.314,Z 862.134,A -85,B 0,C 180,E1 -1344.507,E2 -1344.507} C_VEL
LIN {X 0,Y 587.331,Z 862.13,A -85,B 0,C 180,E1 -1347.257,E2 -1347.257} C_VEL
LIN {X 0,Y 587.382,Z 862.132,A -85,B 0,C 180,E1 -1350,E2 -1350} C_VEL
LIN {X 0,Y 587.338,Z 862.132,A -85,B 0,C 180,E1 -1352.744,E2 -1352.744} C_VEL
LIN {X 0,Y 587.309,Z 862.133,A -85,B 0,C 180,E1 -1355.494,E2 -1355.494} C_VEL
LIN {X 0,Y 587.314,Z 862.139,A -85,B 0,C 180,E1 -1358.256,E2 -1358.256} C_VEL
LIN {X 0,Y 587.303,Z 862.137,A -85,B 0,C 180,E1 -1361.107,E2 -1361.107} C_VEL
LIN {X 0,Y 587.312,Z 862.132,A -85,B 0,C 180,E1 -1363.847,E2 -1363.847} C_VEL
LIN {X 0,Y 587.305,Z 862.143,A -85,B 0,C 180,E1 -1366.798,E2 -1366.798} C_VEL
LIN {X 0,Y 587.291,Z 862.137,A -85,B 0,C 180,E1 -1369.577,E2 -1369.577} C_VEL
LIN {X 0,Y 587.267,Z 862.139,A -85,B 0,C 180,E1 -1371.777,E2 -1371.777} C_VEL
LIN {X 0,Y 587.287,Z 862.137,A -85,B 0,C 180,E1 -1374.565,E2 -1374.565} C_VEL
LIN {X 0,Y 587.303,Z 862.139,A -85,B 0,C 180,E1 -1377.048,E2 -1377.048} C_VEL
LIN {X 0,Y 587.294,Z 862.135,A -85,B 0,C 180,E1 -1380.173,E2 -1380.173} C_VEL
LIN {X 0,Y 587.303,Z 862.133,A -85,B 0,C 180,E1 -1382.582,E2 -1382.582} C_VEL
LIN {X 0,Y 587.292,Z 862.136,A -85,B 0,C 180,E1 -1385.058,E2 -1385.058} C_VEL
LIN {X 0,Y 587.286,Z 862.147,A -85,B 0,C 180,E1 -1387.831,E2 -1387.831} C_VEL
LIN {X 0,Y 587.286,Z 862.141,A -85,B 0,C 180,E1 -1390.257,E2 -1390.257} C_VEL
LIN {X 0,Y 587.277,Z 862.137,A -85,B 0,C 180,E1 -1393.114,E2 -1393.114} C_VEL
LIN {X 0,Y 587.289,Z 862.144,A -85,B 0,C 180,E1 -1396.046,E2 -1396.046} C_VEL
LIN {X 0,Y 587.279,Z 862.138,A -85,B 0,C 180,E1 -1398.932,E2 -1398.932} C_VEL
LIN {X 0,Y 587.268,Z 862.138,A -85,B 0,C 180,E1 -1401.515,E2 -1401.515} C_VEL
LIN {X 0,Y 587.272,Z 862.141,A -85,B 0,C 180,E1 -1404.098,E2 -1404.098} C_VEL
LIN {X 0,Y 587.314,Z 862.143,A -85,B 0,C 180,E1 -1406.601,E2 -1406.601} C_VEL
LIN {X 0,Y 587.287,Z 862.136,A -85,B 0,C 180,E1 -1409.499,E2 -1409.499} C_VEL
LIN {X 0,Y 587.299,Z 862.136,A -85,B 0,C 180,E1 -1412.318,E2 -1412.318} C_VEL
LIN {X 0,Y 587.287,Z 862.143,A -85,B 0,C 180,E1 -1415.238,E2 -1415.238} C_VEL
LIN {X 0,Y 587.301,Z 862.139,A -85,B 0,C 180,E1 -1417.484,E2 -1417.484} C_VEL
LIN {X 0,Y 587.304,Z 862.137,A -85,B 0,C 180,E1 -1419.694,E2 -1419.694} C_VEL
LIN {X 0,Y 587.274,Z 862.139,A -85,B 0,C 180,E1 -1421.871,E2 -1421.871} C_VEL
LIN {X 0,Y 587.285,Z 862.137,A -85,B 0,C 180,E1 -1424.023,E2 -1424.023} C_VEL
LIN {X 0,Y 587.31,Z 862.134,A -85,B 0,C 180,E1 -1426.153,E2 -1426.153} C_VEL
LIN {X 0,Y 587.294,Z 862.136,A -85,B 0,C 180,E1 -1428.961,E2 -1428.961} C_VEL
LIN {X 0,Y 587.314,Z 862.144,A -85,B 0,C 180,E1 -1431.744,E2 -1431.744} C_VEL
LIN {X 0,Y 587.312,Z 862.134,A -85,B 0,C 180,E1 -1434.506,E2 -1434.506} C_VEL
LIN {X 0,Y 587.328,Z 862.131,A -85,B 0,C 180,E1 -1437.256,E2 -1437.256} C_VEL
LIN {X 0,Y 587.38,Z 862.133,A -85,B 0,C 180,E1 -1440,E2 -1440} C_VEL
LIN {X 0,Y 587.336,Z 862.132,A -85,B 0,C 180,E1 -1442.743,E2 -1442.743} C_VEL
LIN {X 0,Y 587.308,Z 862.133,A -85,B 0,C 180,E1 -1445.493,E2 -1445.493} C_VEL
LIN {X 0,Y 587.312,Z 862.139,A -85,B 0,C 180,E1 -1448.256,E2 -1448.256} C_VEL
LIN {X 0,Y 587.3,Z 862.137,A -85,B 0,C 180,E1 -1451.107,E2 -1451.107} C_VEL
LIN {X 0,Y 587.31,Z 862.133,A -85,B 0,C 180,E1 -1453.847,E2 -1453.847} C_VEL
LIN {X 0,Y 587.303,Z 862.144,A -85,B 0,C 180,E1 -1456.798,E2 -1456.798} C_VEL
LIN {X 0,Y 587.289,Z 862.137,A -85,B 0,C 180,E1 -1459.577,E2 -1459.577} C_VEL
LIN {X 0,Y 587.264,Z 862.139,A -85,B 0,C 180,E1 -1461.776,E2 -1461.776} C_VEL
LIN {X 0,Y 587.284,Z 862.137,A -85,B 0,C 180,E1 -1464.565,E2 -1464.565} C_VEL
LIN {X 0,Y 587.301,Z 862.14,A -85,B 0,C 180,E1 -1467.047,E2 -1467.047} C_VEL
LIN {X 0,Y 587.291,Z 862.136,A -85,B 0,C 180,E1 -1470.172,E2 -1470.172} C_VEL
LIN {X 0,Y 587.299,Z 862.134,A -85,B 0,C 180,E1 -1472.581,E2 -1472.581} C_VEL
LIN {X 0,Y 587.29,Z 862.137,A -85,B 0,C 180,E1 -1475.058,E2 -1475.058} C_VEL
LIN {X 0,Y 587.301,Z 862.145,A -85,B 0,C 180,E1 -1477.833,E2 -1477.833} C_VEL
LIN {X 0,Y 587.283,Z 862.141,A -85,B 0,C 180,E1 -1480.257,E2 -1480.257} C_VEL
LIN {X 0,Y 587.274,Z 862.137,A -85,B 0,C 180,E1 -1483.113,E2 -1483.113} C_VEL
LIN {X 0,Y 587.285,Z 862.145,A -85,B 0,C 180,E1 -1486.046,E2 -1486.046} C_VEL
LIN {X 0,Y 587.276,Z 862.138,A -85,B 0,C 180,E1 -1488.932,E2 -1488.932} C_VEL
LIN {X 0,Y 587.266,Z 862.138,A -85,B 0,C 180,E1 -1491.515,E2 -1491.515} C_VEL
LIN {X 0,Y 587.268,Z 862.142,A -85,B 0,C 180,E1 -1494.098,E2 -1494.098} C_VEL
LIN {X 0,Y 587.31,Z 862.144,A -85,B 0,C 180,E1 -1496.601,E2 -1496.601} C_VEL
LIN {X 0,Y 587.284,Z 862.136,A -85,B 0,C 180,E1 -1499.499,E2 -1499.499} C_VEL
LIN {X 0,Y 587.294,Z 862.137,A -85,B 0,C 180,E1 -1502.318,E2 -1502.318} C_VEL
LIN {X 0,Y 587.283,Z 862.144,A -85,B 0,C 180,E1 -1505.238,E2 -1505.238} C_VEL
LIN {X 0,Y 587.299,Z 862.2,A -85,B 0,C 180,E1 -1508.086,E2 -1508.086} C_VEL
LIN {X 0,Y 587.654,Z 867.504,A -85,B 0,C 180,E1 -1508.974,E2 -1508.974} C_VEL
LIN {X 0,Y 587.526,Z 885.369,A -85,B 0,C 180,E1 -1511.88,E2 -1511.88} C_VEL
LIN {X 0,Y 587.395,Z 902.118,A -85,B 0,C 180,E1 -1514.561,E2 -1514.561} C_VEL
LIN {X 0,Y 587.319,Z 919.983,A -85,B 0,C 180,E1 -1517.386,E2 -1517.386} C_VEL
LIN {X 0,Y 587.291,Z 932.754,A -85,B 0,C 180,E1 -1519.387,E2 -1519.387} C_VEL
LIN {X 0,Y 587.568,Z 940.651,A -85,B 0,C 180,E1 -1519.49,E2 -1519.49} C_VEL
LIN {X 0,Y 587.524,Z 1010.431,A -85,B 0,C 180,E1 -1520.359,E2 -1520.359} C_VEL
LIN {X 0,Y 587.486,Z 1020.898,A -85,B 0,C 180,E1 -1520.597,E2 -1520.597} C_VEL
LIN {X 0,Y 587.435,Z 1031.611,A -85,B 0,C 180,E1 -1520.966,E2 -1520.966} C_VEL
LIN {X 0,Y 587.416,Z 1042.234,A -85,B 0,C 180,E1 -1521.485,E2 -1521.485} C_VEL
LIN {X 0,Y 587.343,Z 1050.543,A -85,B 0,C 180,E1 -1522.004,E2 -1522.004} C_VEL
LIN {X 0,Y 587.292,Z 1058.4,A -85,B 0,C 180,E1 -1522.609,E2 -1522.609} C_VEL
LIN {X 0,Y 587.286,Z 1065.164,A -85,B 0,C 180,E1 -1523.241,E2 -1523.241} C_VEL
LIN {X 0,Y 587.265,Z 1071.779,A -85,B 0,C 180,E1 -1523.989,E2 -1523.989} C_VEL
LIN {X 0,Y 587.203,Z 1079.027,A -85,B 0,C 180,E1 -1525.022,E2 -1525.022} C_VEL
LIN {X 0,Y 587.18,Z 1083.63,A -85,B 0,C 180,E1 -1525.882,E2 -1525.882} C_VEL
LIN {X 0,Y 587.192,Z 1086.621,A -85,B 0,C 180,E1 -1526.569,E2 -1526.569} C_VEL
LIN {X 0,Y 587.135,Z 1088.932,A -85,B 0,C 180,E1 -1527.255,E2 -1527.255} C_VEL
LIN {X 0,Y 587.14,Z 1090.679,A -85,B 0,C 180,E1 -1527.942,E2 -1527.942} C_VEL
LIN {X 0,Y 587.145,Z 1091.935,A -85,B 0,C 180,E1 -1528.628,E2 -1528.628} C_VEL
LIN {X 0,Y 587.136,Z 1092.713,A -85,B 0,C 180,E1 -1529.314,E2 -1529.314} C_VEL
LIN {X 0,Y 587.134,Z 1093,A -85,B 0,C 180,E1 -1530,E2 -1530} C_VEL
LIN {X 0,Y 587.136,Z 1092.713,A -85,B 0,C 180,E1 -1530.686,E2 -1530.686} C_VEL
LIN {X 0,Y 587.145,Z 1091.935,A -85,B 0,C 180,E1 -1531.372,E2 -1531.372} C_VEL
LIN {X 0,Y 587.14,Z 1090.679,A -85,B 0,C 180,E1 -1532.058,E2 -1532.058} C_VEL
LIN {X 0,Y 587.155,Z 1087.787,A -85,B 0,C 180,E1 -1533.088,E2 -1533.088} C_VEL
LIN {X 0,Y 587.21,Z 1085.147,A -85,B 0,C 180,E1 -1533.774,E2 -1533.774} C_VEL
LIN {X 0,Y 587.185,Z 1079.986,A -85,B 0,C 180,E1 -1534.806,E2 -1534.806} C_VEL
LIN {X 0,Y 587.238,Z 1074.431,A -85,B 0,C 180,E1 -1535.666,E2 -1535.666} C_VEL
LIN {X 0,Y 587.269,Z 1066.286,A -85,B 0,C 180,E1 -1536.646,E2 -1536.646} C_VEL
LIN {X 0,Y 587.288,Z 1059.418,A -85,B 0,C 180,E1 -1537.305,E2 -1537.305} C_VEL
LIN {X 0,Y 587.33,Z 1051.766,A -85,B 0,C 180,E1 -1537.909,E2 -1537.909} C_VEL
LIN {X 0,Y 587.398,Z 1043.726,A -85,B 0,C 180,E1 -1538.428,E2 -1538.428} C_VEL
LIN {X 0,Y 587.41,Z 1035.396,A -85,B 0,C 180,E1 -1538.861,E2 -1538.861} C_VEL
LIN {X 0,Y 587.425,Z 1026.893,A -85,B 0,C 180,E1 -1539.208,E2 -1539.208} C_VEL
LIN {X 0,Y 587.498,Z 1017.588,A -85,B 0,C 180,E1 -1539.489,E2 -1539.489} C_VEL
LIN {X 0,Y 587.538,Z 1006.552,A -85,B 0,C 180,E1 -1539.706,E2 -1539.706} C_VEL
LIN {X 0,Y 587.433,Z 933.852,A -85,B 0,C 180,E1 -1540.595,E2 -1540.595} C_VEL
LIN {X 0,Y 587.273,Z 932.686,A -85,B 0,C 180,E1 -1540.624,E2 -1540.624} C_VEL
LIN {X 0,Y 587.343,Z 914.402,A -85,B 0,C 180,E1 -1543.493,E2 -1543.493} C_VEL
LIN {X 0,Y 587.459,Z 897.653,A -85,B 0,C 180,E1 -1546.15,E2 -1546.15} C_VEL
LIN {X 0,Y 587.559,Z 880.904,A -85,B 0,C 180,E1 -1548.842,E2 -1548.842} C_VEL
LIN {X 0,Y 587.619,Z 865.274,A -85,B 0,C 180,E1 -1551.394,E2 -1551.394} C_VEL
LIN {X 0,Y 587.286,Z 862.142,A -85,B 0,C 180,E1 -1551.96,E2 -1551.96} C_VEL
LIN {X 0,Y 587.282,Z 862.144,A -85,B 0,C 180,E1 -1554.762,E2 -1554.762} C_VEL
LIN {X 0,Y 587.293,Z 862.138,A -85,B 0,C 180,E1 -1557.682,E2 -1557.682} C_VEL
LIN {X 0,Y 587.282,Z 862.137,A -85,B 0,C 180,E1 -1560.501,E2 -1560.501} C_VEL
LIN {X 0,Y 587.308,Z 862.145,A -85,B 0,C 180,E1 -1563.398,E2 -1563.398} C_VEL
LIN {X 0,Y 587.267,Z 862.142,A -85,B 0,C 180,E1 -1565.902,E2 -1565.902} C_VEL
LIN {X 0,Y 587.264,Z 862.139,A -85,B 0,C 180,E1 -1568.484,E2 -1568.484} C_VEL
LIN {X 0,Y 587.279,Z 862.139,A -85,B 0,C 180,E1 -1571.162,E2 -1571.162} C_VEL
LIN {X 0,Y 587.283,Z 862.143,A -85,B 0,C 180,E1 -1574.109,E2 -1574.109} C_VEL
LIN {X 0,Y 587.266,Z 862.138,A -85,B 0,C 180,E1 -1576.989,E2 -1576.989} C_VEL
LIN {X 0,Y 587.287,Z 862.144,A -85,B 0,C 180,E1 -1579.986,E2 -1579.986} C_VEL
LIN {X 0,Y 587.304,Z 862.142,A -85,B 0,C 180,E1 -1582.39,E2 -1582.39} C_VEL
LIN {X 0,Y 587.315,Z 862.133,A -85,B 0,C 180,E1 -1585.657,E2 -1585.657} C_VEL
LIN {X 0,Y 587.297,Z 862.141,A -85,B 0,C 180,E1 -1588.229,E2 -1588.229} C_VEL
LIN {X 0,Y 587.295,Z 862.141,A -85,B 0,C 180,E1 -1590.876,E2 -1590.876} C_VEL
LIN {X 0,Y 587.292,Z 862.135,A -85,B 0,C 180,E1 -1593.833,E2 -1593.833} C_VEL
LIN {X 0,Y 587.277,Z 862.146,A -85,B 0,C 180,E1 -1596.74,E2 -1596.74} C_VEL
LIN {X 0,Y 587.295,Z 862.136,A -85,B 0,C 180,E1 -1599.694,E2 -1599.694} C_VEL
LIN {X 0,Y 587.271,Z 862.139,A -85,B 0,C 180,E1 -1602.232,E2 -1602.232} C_VEL
LIN {X 0,Y 587.329,Z 862.238,A -85,B 0,C 180,E1 -1602.594,E2 -1602.594} C_VEL
LIN {X 0,Y 587.277,Z 875.602,A -85,B 0,C 180,E1 -1605.445,E2 -1605.445} C_VEL
LIN {X 0,Y 587.239,Z 887.297,A -85,B 0,C 180,E1 -1607.911,E2 -1607.911} C_VEL
LIN {X 0,Y 587.231,Z 894.67,A -85,B 0,C 180,E1 -1609.454,E2 -1609.454} C_VEL
LIN {X 0,Y 587.58,Z 902.465,A -85,B 0,C 180,E1 -1609.557,E2 -1609.557} C_VEL
LIN {X 0,Y 587.501,Z 970.369,A -85,B 0,C 180,E1 -1610.403,E2 -1610.403} C_VEL
LIN {X 0,Y 587.466,Z 980.861,A -85,B 0,C 180,E1 -1610.641,E2 -1610.641} C_VEL
LIN {X 0,Y 587.406,Z 992.566,A -85,B 0,C 180,E1 -1611.052,E2 -1611.052} C_VEL
LIN {X 0,Y 587.401,Z 1002.983,A -85,B 0,C 180,E1 -1611.572,E2 -1611.572} C_VEL
LIN {X 0,Y 587.333,Z 1011.159,A -85,B 0,C 180,E1 -1612.091,E2 -1612.091} C_VEL
LIN {X 0,Y 587.289,Z 1018.905,A -85,B 0,C 180,E1 -1612.695,E2 -1612.695} C_VEL
LIN {X 0,Y 587.286,Z 1026.736,A -85,B 0,C 180,E1 -1613.443,E2 -1613.443} C_VEL
LIN {X 0,Y 587.238,Z 1034.135,A -85,B 0,C 180,E1 -1614.334,E2 -1614.334} C_VEL
LIN {X 0,Y 587.184,Z 1039.751,A -85,B 0,C 180,E1 -1615.194,E2 -1615.194} C_VEL
LIN {X 0,Y 587.21,Z 1044.968,A -85,B 0,C 180,E1 -1616.226,E2 -1616.226} C_VEL
LIN {X 0,Y 587.135,Z 1048.793,A -85,B 0,C 180,E1 -1617.256,E2 -1617.256} C_VEL
LIN {X 0,Y 587.14,Z 1050.587,A -85,B 0,C 180,E1 -1617.942,E2 -1617.942} C_VEL
LIN {X 0,Y 587.144,Z 1051.887,A -85,B 0,C 180,E1 -1618.629,E2 -1618.629} C_VEL
LIN {X 0,Y 587.136,Z 1052.704,A -85,B 0,C 180,E1 -1619.314,E2 -1619.314} C_VEL
LIN {X 0,Y 587.135,Z 1052.996,A -85,B 0,C 180,E1 -1620,E2 -1620} C_VEL
LIN {X 0,Y 587.137,Z 1052.745,A -85,B 0,C 180,E1 -1620.686,E2 -1620.686} C_VEL
LIN {X 0,Y 587.146,Z 1052.01,A -85,B 0,C 180,E1 -1621.372,E2 -1621.372} C_VEL
LIN {X 0,Y 587.141,Z 1050.795,A -85,B 0,C 180,E1 -1622.058,E2 -1622.058} C_VEL
LIN {X 0,Y 587.156,Z 1047.947,A -85,B 0,C 180,E1 -1623.088,E2 -1623.088} C_VEL
LIN {X 0,Y 587.182,Z 1043.846,A -85,B 0,C 180,E1 -1624.119,E2 -1624.119} C_VEL
LIN {X 0,Y 587.171,Z 1038.256,A -85,B 0,C 180,E1 -1625.151,E2 -1625.151} C_VEL
LIN {X 0,Y 587.264,Z 1032.17,A -85,B 0,C 180,E1 -1626.011,E2 -1626.011} C_VEL
LIN {X 0,Y 587.286,Z 1025.638,A -85,B 0,C 180,E1 -1626.758,E2 -1626.758} C_VEL
LIN {X 0,Y 587.31,Z 1017.924,A -85,B 0,C 180,E1 -1627.478,E2 -1627.478} C_VEL
LIN {X 0,Y 587.35,Z 1008.749,A -85,B 0,C 180,E1 -1628.169,E2 -1628.169} C_VEL
LIN {X 0,Y 587.433,Z 998.21,A -85,B 0,C 180,E1 -1628.775,E2 -1628.775} C_VEL
LIN {X 0,Y 587.412,Z 988.133,A -85,B 0,C 180,E1 -1629.209,E2 -1629.209} C_VEL
LIN {X 0,Y 587.453,Z 979.296,A -85,B 0,C 180,E1 -1629.49,E2 -1629.49} C_VEL
LIN {X 0,Y 587.5,Z 970.516,A -85,B 0,C 180,E1 -1629.685,E2 -1629.685} C_VEL
LIN {X 0,Y 587.591,Z 910.793,A -85,B 0,C 180,E1 -1630.431,E2 -1630.431} C_VEL
LIN {X 0,Y 586.948,Z 906.597,A -85,B 0,C 180,E1 -1630.496,E2 -1630.496} C_VEL
LIN {X 0,Y 585.331,Z 902.639,A -85,B 0,C 180,E1 -1630.572,E2 -1630.572} C_VEL
LIN {X 0,Y 583.322,Z 899.008,A -85,B 0,C 180,E1 -1630.668,E2 -1630.668} C_VEL
LIN {X 0,Y 581.209,Z 895.311,A -85,B 0,C 180,E1 -1630.878,E2 -1630.878} C_VEL
LIN {X 0,Y 580.24,Z 892.997,A -85,B 0,C 180,E1 -1631.134,E2 -1631.134} C_VEL
LIN {X 0,Y 580.178,Z 892.53,A -85,B 0,C 180,E1 -1631.219,E2 -1631.219} C_VEL
LIN {X 0,Y 580.202,Z 879.364,A -85,B 0,C 180,E1 -1634.02,E2 -1634.02} C_VEL
LIN {X 0,Y 580.316,Z 865.917,A -85,B 0,C 180,E1 -1636.914,E2 -1636.914} C_VEL
LIN {X 0,Y 580.263,Z 863.014,A -85,B 0,C 180,E1 -1637.576,E2 -1637.576} C_VEL
LIN {X 0,Y 580.251,Z 863.012,A -85,B 0,C 180,E1 -1639.825,E2 -1639.825} C_VEL
LIN {X 0,Y 580.211,Z 863.017,A -85,B 0,C 180,E1 -1642.056,E2 -1642.056} C_VEL
LIN {X 0,Y 580.247,Z 863.015,A -85,B 0,C 180,E1 -1644.714,E2 -1644.714} C_VEL
LIN {X 0,Y 580.25,Z 863.023,A -85,B 0,C 180,E1 -1647.404,E2 -1647.404} C_VEL
LIN {X 0,Y 580.247,Z 863.018,A -85,B 0,C 180,E1 -1649.776,E2 -1649.776} C_VEL
LIN {X 0,Y 580.276,Z 863.011,A -85,B 0,C 180,E1 -1652.202,E2 -1652.202} C_VEL
LIN {X 0,Y 580.269,Z 863.01,A -85,B 0,C 180,E1 -1654.698,E2 -1654.698} C_VEL
LIN {X 0,Y 580.26,Z 863.013,A -85,B 0,C 180,E1 -1657.272,E2 -1657.272} C_VEL
LIN {X 0,Y 580.248,Z 863.018,A -85,B 0,C 180,E1 -1660.265,E2 -1660.265} C_VEL
LIN {X 0,Y 580.244,Z 863.014,A -85,B 0,C 180,E1 -1662.71,E2 -1662.71} C_VEL
LIN {X 0,Y 580.238,Z 863.016,A -85,B 0,C 180,E1 -1665.613,E2 -1665.613} C_VEL
LIN {X 0,Y 580.234,Z 863.024,A -85,B 0,C 180,E1 -1668.227,E2 -1668.227} C_VEL
LIN {X 0,Y 580.238,Z 863.016,A -85,B 0,C 180,E1 -1670.962,E2 -1670.962} C_VEL
LIN {X 0,Y 580.232,Z 863.014,A -85,B 0,C 180,E1 -1673.594,E2 -1673.594} C_VEL
LIN {X 0,Y 580.267,Z 863.013,A -85,B 0,C 180,E1 -1676.142,E2 -1676.142} C_VEL
LIN {X 0,Y 580.241,Z 863.022,A -85,B 0,C 180,E1 -1678.612,E2 -1678.612} C_VEL
LIN {X 0,Y 580.246,Z 863.021,A -85,B 0,C 180,E1 -1681.021,E2 -1681.021} C_VEL
LIN {X 0,Y 580.253,Z 863.013,A -85,B 0,C 180,E1 -1683.675,E2 -1683.675} C_VEL
LIN {X 0,Y 580.239,Z 863.015,A -85,B 0,C 180,E1 -1686.44,E2 -1686.44} C_VEL
LIN {X 0,Y 580.262,Z 863.018,A -85,B 0,C 180,E1 -1689.437,E2 -1689.437} C_VEL
LIN {X 0,Y 580.238,Z 863.019,A -85,B 0,C 180,E1 -1691.644,E2 -1691.644} C_VEL
LIN {X 0,Y 580.246,Z 863.017,A -85,B 0,C 180,E1 -1693.825,E2 -1693.825} C_VEL
LIN {X 0,Y 580.29,Z 863.011,A -85,B 0,C 180,E1 -1695.982,E2 -1695.982} C_VEL
LIN {X 0,Y 580.273,Z 863.009,A -85,B 0,C 180,E1 -1698.826,E2 -1698.826} C_VEL
LIN {X 0,Y 580.289,Z 863.016,A -85,B 0,C 180,E1 -1701.643,E2 -1701.643} C_VEL
LIN {X 0,Y 580.284,Z 863.01,A -85,B 0,C 180,E1 -1704.44,E2 -1704.44} C_VEL
LIN {X 0,Y 580.299,Z 863.006,A -85,B 0,C 180,E1 -1707.223,E2 -1707.223} C_VEL
LIN {X 0,Y 580.351,Z 863.008,A -85,B 0,C 180,E1 -1710,E2 -1710} C_VEL
LIN {X 0,Y 580.305,Z 863.008,A -85,B 0,C 180,E1 -1712.777,E2 -1712.777} C_VEL
LIN {X 0,Y 580.28,Z 863.009,A -85,B 0,C 180,E1 -1715.56,E2 -1715.56} C_VEL
LIN {X 0,Y 580.288,Z 863.016,A -85,B 0,C 180,E1 -1718.357,E2 -1718.357} C_VEL
LIN {X 0,Y 580.273,Z 863.012,A -85,B 0,C 180,E1 -1721.174,E2 -1721.174} C_VEL
LIN {X 0,Y 580.276,Z 863.009,A -85,B 0,C 180,E1 -1724.018,E2 -1724.018} C_VEL
LIN {X 0,Y 580.274,Z 863.021,A -85,B 0,C 180,E1 -1726.899,E2 -1726.899} C_VEL
LIN {X 0,Y 580.252,Z 863.012,A -85,B 0,C 180,E1 -1729.824,E2 -1729.824} C_VEL
LIN {X 0,Y 580.211,Z 863.017,A -85,B 0,C 180,E1 -1732.055,E2 -1732.055} C_VEL
LIN {X 0,Y 580.243,Z 863.016,A -85,B 0,C 180,E1 -1734.712,E2 -1734.712} C_VEL
LIN {X 0,Y 580.248,Z 863.023,A -85,B 0,C 180,E1 -1737.404,E2 -1737.404} C_VEL
LIN {X 0,Y 580.249,Z 863.018,A -85,B 0,C 180,E1 -1739.775,E2 -1739.775} C_VEL
LIN {X 0,Y 580.242,Z 863.015,A -85,B 0,C 180,E1 -1742.204,E2 -1742.204} C_VEL
LIN {X 0,Y 580.27,Z 863.009,A -85,B 0,C 180,E1 -1744.698,E2 -1744.698} C_VEL
LIN {X 0,Y 580.258,Z 863.014,A -85,B 0,C 180,E1 -1747.272,E2 -1747.272} C_VEL
LIN {X 0,Y 580.249,Z 863.017,A -85,B 0,C 180,E1 -1750.265,E2 -1750.265} C_VEL
LIN {X 0,Y 580.243,Z 863.014,A -85,B 0,C 180,E1 -1752.71,E2 -1752.71} C_VEL
LIN {X 0,Y 580.237,Z 863.016,A -85,B 0,C 180,E1 -1755.613,E2 -1755.613} C_VEL
LIN {X 0,Y 580.235,Z 863.025,A -85,B 0,C 180,E1 -1758.227,E2 -1758.227} C_VEL
LIN {X 0,Y 580.238,Z 863.016,A -85,B 0,C 180,E1 -1760.961,E2 -1760.961} C_VEL
LIN {X 0,Y 580.222,Z 863.016,A -85,B 0,C 180,E1 -1763.592,E2 -1763.592} C_VEL
LIN {X 0,Y 580.267,Z 863.013,A -85,B 0,C 180,E1 -1766.141,E2 -1766.141} C_VEL
LIN {X 0,Y 580.241,Z 863.022,A -85,B 0,C 180,E1 -1768.612,E2 -1768.612} C_VEL
LIN {X 0,Y 580.245,Z 863.021,A -85,B 0,C 180,E1 -1771.021,E2 -1771.021} C_VEL
LIN {X 0,Y 580.253,Z 863.013,A -85,B 0,C 180,E1 -1773.675,E2 -1773.675} C_VEL
LIN {X 0,Y 580.238,Z 863.015,A -85,B 0,C 180,E1 -1776.44,E2 -1776.44} C_VEL
LIN {X 0,Y 580.26,Z 863.018,A -85,B 0,C 180,E1 -1779.436,E2 -1779.436} C_VEL
LIN {X 0,Y 580.236,Z 863.019,A -85,B 0,C 180,E1 -1781.644,E2 -1781.644} C_VEL
LIN {X 0,Y 580.244,Z 863.017,A -85,B 0,C 180,E1 -1783.824,E2 -1783.824} C_VEL
LIN {X 0,Y 580.275,Z 863.012,A -85,B 0,C 180,E1 -1785.981,E2 -1785.981} C_VEL
LIN {X 0,Y 580.272,Z 863.01,A -85,B 0,C 180,E1 -1788.826,E2 -1788.826} C_VEL
LIN {X 0,Y 580.287,Z 863.017,A -85,B 0,C 180,E1 -1791.643,E2 -1791.643} C_VEL
LIN {X 0,Y 580.282,Z 863.01,A -85,B 0,C 180,E1 -1794.439,E2 -1794.439} C_VEL
LIN {X 0,Y 580.296,Z 863.007,A -85,B 0,C 180,E1 -1797.223,E2 -1797.223} C_VEL
LIN {X 0,Y 580.349,Z 863.009,A -85,B 0,C 180,E1 -1800,E2 -1800} C_VEL
LIN {X 0,Y 580.302,Z 863.008,A -85,B 0,C 180,E1 -1802.776,E2 -1802.776} C_VEL
LIN {X 0,Y 580.278,Z 863.009,A -85,B 0,C 180,E1 -1805.56,E2 -1805.56} C_VEL
LIN {X 0,Y 580.286,Z 863.016,A -85,B 0,C 180,E1 -1808.356,E2 -1808.356} C_VEL
LIN {X 0,Y 580.27,Z 863.012,A -85,B 0,C 180,E1 -1811.174,E2 -1811.174} C_VEL
LIN {X 0,Y 580.273,Z 863.01,A -85,B 0,C 180,E1 -1814.018,E2 -1814.018} C_VEL
LIN {X 0,Y 580.27,Z 863.021,A -85,B 0,C 180,E1 -1816.898,E2 -1816.898} C_VEL
LIN {X 0,Y 580.249,Z 863.012,A -85,B 0,C 180,E1 -1819.824,E2 -1819.824} C_VEL
LIN {X 0,Y 580.209,Z 863.017,A -85,B 0,C 180,E1 -1822.055,E2 -1822.055} C_VEL
LIN {X 0,Y 580.24,Z 863.016,A -85,B 0,C 180,E1 -1824.712,E2 -1824.712} C_VEL
LIN {X 0,Y 580.245,Z 863.023,A -85,B 0,C 180,E1 -1827.404,E2 -1827.404} C_VEL
LIN {X 0,Y 580.245,Z 863.018,A -85,B 0,C 180,E1 -1829.775,E2 -1829.775} C_VEL
LIN {X 0,Y 580.239,Z 863.015,A -85,B 0,C 180,E1 -1832.204,E2 -1832.204} C_VEL
LIN {X 0,Y 580.267,Z 863.01,A -85,B 0,C 180,E1 -1834.698,E2 -1834.698} C_VEL
LIN {X 0,Y 580.257,Z 863.014,A -85,B 0,C 180,E1 -1837.271,E2 -1837.271} C_VEL
LIN {X 0,Y 580.245,Z 863.017,A -85,B 0,C 180,E1 -1840.265,E2 -1840.265} C_VEL
LIN {X 0,Y 580.24,Z 863.014,A -85,B 0,C 180,E1 -1842.71,E2 -1842.71} C_VEL
LIN {X 0,Y 580.235,Z 863.016,A -85,B 0,C 180,E1 -1845.612,E2 -1845.612} C_VEL
LIN {X 0,Y 580.231,Z 863.026,A -85,B 0,C 180,E1 -1848.226,E2 -1848.226} C_VEL
LIN {X 0,Y 580.235,Z 863.016,A -85,B 0,C 180,E1 -1850.961,E2 -1850.961} C_VEL
LIN {X 0,Y 580.218,Z 863.016,A -85,B 0,C 180,E1 -1853.592,E2 -1853.592} C_VEL
LIN {X 0,Y 580.263,Z 863.014,A -85,B 0,C 180,E1 -1856.141,E2 -1856.141} C_VEL
LIN {X 0,Y 580.237,Z 863.023,A -85,B 0,C 180,E1 -1858.612,E2 -1858.612} C_VEL
LIN {X 0,Y 580.241,Z 863.021,A -85,B 0,C 180,E1 -1861.021,E2 -1861.021} C_VEL
LIN {X 0,Y 580.248,Z 863.014,A -85,B 0,C 180,E1 -1863.675,E2 -1863.675} C_VEL
LIN {X 0,Y 580.238,Z 863.017,A -85,B 0,C 180,E1 -1866.44,E2 -1866.44} C_VEL
LIN {X 0,Y 580.242,Z 863.037,A -85,B 0,C 180,E1 -1867.946,E2 -1867.946} C_VEL
LIN {X 0,Y 580.71,Z 868.25,A -85,B 0,C 180,E1 -1868.835,E2 -1868.835} C_VEL
LIN {X 0,Y 580.538,Z 885.369,A -85,B 0,C 180,E1 -1871.654,E2 -1871.654} C_VEL
LIN {X 0,Y 580.409,Z 902.118,A -85,B 0,C 180,E1 -1874.37,E2 -1874.37} C_VEL
LIN {X 0,Y 580.28,Z 921.099,A -85,B 0,C 180,E1 -1877.408,E2 -1877.408} C_VEL
LIN {X 0,Y 580.213,Z 932.737,A -85,B 0,C 180,E1 -1879.253,E2 -1879.253} C_VEL
LIN {X 0,Y 580.613,Z 937.226,A -85,B 0,C 180,E1 -1879.32,E2 -1879.32} C_VEL
LIN {X 0,Y 580.547,Z 1010.43,A -85,B 0,C 180,E1 -1880.242,E2 -1880.242} C_VEL
LIN {X 0,Y 580.477,Z 1020.068,A -85,B 0,C 180,E1 -1880.461,E2 -1880.461} C_VEL
LIN {X 0,Y 580.426,Z 1031.61,A -85,B 0,C 180,E1 -1880.856,E2 -1880.856} C_VEL
LIN {X 0,Y 580.392,Z 1042.234,A -85,B 0,C 180,E1 -1881.382,E2 -1881.382} C_VEL
LIN {X 0,Y 580.303,Z 1050.544,A -85,B 0,C 180,E1 -1881.906,E2 -1881.906} C_VEL
LIN {X 0,Y 580.25,Z 1058.4,A -85,B 0,C 180,E1 -1882.518,E2 -1882.518} C_VEL
LIN {X 0,Y 580.227,Z 1065.463,A -85,B 0,C 180,E1 -1883.189,E2 -1883.189} C_VEL
LIN {X 0,Y 580.193,Z 1073.189,A -85,B 0,C 180,E1 -1884.09,E2 -1884.09} C_VEL
LIN {X 0,Y 580.102,Z 1079.027,A -85,B 0,C 180,E1 -1884.961,E2 -1884.961} C_VEL
LIN {X 0,Y 580.105,Z 1083.63,A -85,B 0,C 180,E1 -1885.831,E2 -1885.831} C_VEL
LIN {X 0,Y 580.121,Z 1086.621,A -85,B 0,C 180,E1 -1886.527,E2 -1886.527} C_VEL
LIN {X 0,Y 580.046,Z 1088.932,A -85,B 0,C 180,E1 -1887.222,E2 -1887.222} C_VEL
LIN {X 0,Y 580.04,Z 1090.679,A -85,B 0,C 180,E1 -1887.917,E2 -1887.917} C_VEL
LIN {X 0,Y 580.045,Z 1091.935,A -85,B 0,C 180,E1 -1888.611,E2 -1888.611} C_VEL
LIN {X 0,Y 580.036,Z 1092.712,A -85,B 0,C 180,E1 -1889.306,E2 -1889.306} C_VEL
LIN {X 0,Y 580.034,Z 1093,A -85,B 0,C 180,E1 -1890,E2 -1890} C_VEL
LIN {X 0,Y 580.036,Z 1092.712,A -85,B 0,C 180,E1 -1890.694,E2 -1890.694} C_VEL
LIN {X 0,Y 580.045,Z 1091.935,A -85,B 0,C 180,E1 -1891.388,E2 -1891.388} C_VEL
LIN {X 0,Y 580.04,Z 1090.68,A -85,B 0,C 180,E1 -1892.083,E2 -1892.083} C_VEL
LIN {X 0,Y 580.07,Z 1087.788,A -85,B 0,C 180,E1 -1893.125,E2 -1893.125} C_VEL
LIN {X 0,Y 580.137,Z 1085.147,A -85,B 0,C 180,E1 -1893.82,E2 -1893.82} C_VEL
LIN {X 0,Y 580.096,Z 1079.986,A -85,B 0,C 180,E1 -1894.865,E2 -1894.865} C_VEL
LIN {X 0,Y 580.173,Z 1074.431,A -85,B 0,C 180,E1 -1895.735,E2 -1895.735} C_VEL
LIN {X 0,Y 580.209,Z 1066.947,A -85,B 0,C 180,E1 -1896.659,E2 -1896.659} C_VEL
LIN {X 0,Y 580.237,Z 1059.419,A -85,B 0,C 180,E1 -1897.394,E2 -1897.394} C_VEL
LIN {X 0,Y 580.284,Z 1051.767,A -85,B 0,C 180,E1 -1898.006,E2 -1898.006} C_VEL
LIN {X 0,Y 580.371,Z 1043.728,A -85,B 0,C 180,E1 -1898.531,E2 -1898.531} C_VEL
LIN {X 0,Y 580.401,Z 1035.398,A -85,B 0,C 180,E1 -1898.969,E2 -1898.969} C_VEL
LIN {X 0,Y 580.431,Z 1026.894,A -85,B 0,C 180,E1 -1899.32,E2 -1899.32} C_VEL
LIN {X 0,Y 580.471,Z 1017.588,A -85,B 0,C 180,E1 -1899.605,E2 -1899.605} C_VEL
LIN {X 0,Y 580.54,Z 1006.552,A -85,B 0,C 180,E1 -1899.824,E2 -1899.824} C_VEL
LIN {X 0,Y 580.466,Z 934.692,A -85,B 0,C 180,E1 -1900.714,E2 -1900.714} C_VEL
LIN {X 0,Y 580.214,Z 932.727,A -85,B 0,C 180,E1 -1900.749,E2 -1900.749} C_VEL
LIN {X 0,Y 580.32,Z 914.402,A -85,B 0,C 180,E1 -1903.66,E2 -1903.66} C_VEL
LIN {X 0,Y 580.48,Z 896.536,A -85,B 0,C 180,E1 -1906.53,E2 -1906.53} C_VEL
LIN {X 0,Y 580.598,Z 878.524,A -85,B 0,C 180,E1 -1909.468,E2 -1909.468} C_VEL
LIN {X 0,Y 580.61,Z 865.272,A -85,B 0,C 180,E1 -1911.665,E2 -1911.665} C_VEL
LIN {X 0,Y 580.246,Z 863.02,A -85,B 0,C 180,E1 -1912.077,E2 -1912.077} C_VEL
LIN {X 0,Y 580.229,Z 863.026,A -85,B 0,C 180,E1 -1915.083,E2 -1915.083} C_VEL
LIN {X 0,Y 580.236,Z 863.016,A -85,B 0,C 180,E1 -1917.847,E2 -1917.847} C_VEL
LIN {X 0,Y 580.236,Z 863.016,A -85,B 0,C 180,E1 -1920.687,E2 -1920.687} C_VEL
LIN {X 0,Y 580.269,Z 863.021,A -85,B 0,C 180,E1 -1923.311,E2 -1923.311} C_VEL
LIN {X 0,Y 580.218,Z 863.023,A -85,B 0,C 180,E1 -1925.753,E2 -1925.753} C_VEL
LIN {X 0,Y 580.231,Z 863.017,A -85,B 0,C 180,E1 -1928.151,E2 -1928.151} C_VEL
LIN {X 0,Y 580.227,Z 863.015,A -85,B 0,C 180,E1 -1930.85,E2 -1930.85} C_VEL
LIN {X 0,Y 580.22,Z 863.024,A -85,B 0,C 180,E1 -1933.663,E2 -1933.663} C_VEL
LIN {X 0,Y 580.218,Z 863.018,A -85,B 0,C 180,E1 -1936.616,E2 -1936.616} C_VEL
LIN {X 0,Y 580.233,Z 863.014,A -85,B 0,C 180,E1 -1939.151,E2 -1939.151} C_VEL
LIN {X 0,Y 580.243,Z 863.019,A -85,B 0,C 180,E1 -1941.933,E2 -1941.933} C_VEL
LIN {X 0,Y 580.219,Z 863.025,A -85,B 0,C 180,E1 -1944.451,E2 -1944.451} C_VEL
LIN {X 0,Y 580.239,Z 863.016,A -85,B 0,C 180,E1 -1946.972,E2 -1946.972} C_VEL
LIN {X 0,Y 580.246,Z 863.013,A -85,B 0,C 180,E1 -1949.422,E2 -1949.422} C_VEL
LIN {X 0,Y 580.235,Z 863.017,A -85,B 0,C 180,E1 -1952.153,E2 -1952.153} C_VEL
LIN {X 0,Y 580.23,Z 863.025,A -85,B 0,C 180,E1 -1954.917,E2 -1954.917} C_VEL
LIN {X 0,Y 580.245,Z 863.02,A -85,B 0,C 180,E1 -1957.196,E2 -1957.196} C_VEL
LIN {X 0,Y 580.246,Z 863.018,A -85,B 0,C 180,E1 -1959.436,E2 -1959.436} C_VEL
LIN {X 0,Y 580.233,Z 863.019,A -85,B 0,C 180,E1 -1961.644,E2 -1961.644} C_VEL
LIN {X 0,Y 580.288,Z 863.16,A -85,B 0,C 180,E1 -1962.576,E2 -1962.576} C_VEL
LIN {X 0,Y 580.257,Z 875.605,A -85,B 0,C 180,E1 -1965.265,E2 -1965.265} C_VEL
LIN {X 0,Y 580.18,Z 888.97,A -85,B 0,C 180,E1 -1968.116,E2 -1968.116} C_VEL
LIN {X 0,Y 580.157,Z 894.66,A -85,B 0,C 180,E1 -1969.321,E2 -1969.321} C_VEL
LIN {X 0,Y 580.622,Z 902.072,A -85,B 0,C 180,E1 -1969.425,E2 -1969.425} C_VEL
LIN {X 0,Y 580.525,Z 970.402,A -85,B 0,C 180,E1 -1970.286,E2 -1970.286} C_VEL
LIN {X 0,Y 580.463,Z 980.884,A -85,B 0,C 180,E1 -1970.527,E2 -1970.527} C_VEL
LIN {X 0,Y 580.383,Z 992.575,A -85,B 0,C 180,E1 -1970.943,E2 -1970.943} C_VEL
LIN {X 0,Y 580.379,Z 1003.001,A -85,B 0,C 180,E1 -1971.47,E2 -1971.47} C_VEL
LIN {X 0,Y 580.285,Z 1012.393,A -85,B 0,C 180,E1 -1972.082,E2 -1972.082} C_VEL
LIN {X 0,Y 580.245,Z 1021.887,A -85,B 0,C 180,E1 -1972.869,E2 -1972.869} C_VEL
LIN {X 0,Y 580.194,Z 1030.021,A -85,B 0,C 180,E1 -1973.742,E2 -1973.742} C_VEL
LIN {X 0,Y 580.121,Z 1036.5,A -85,B 0,C 180,E1 -1974.613,E2 -1974.613} C_VEL
LIN {X 0,Y 580.122,Z 1041.673,A -85,B 0,C 180,E1 -1975.484,E2 -1975.484} C_VEL
LIN {X 0,Y 580.121,Z 1046.439,A -85,B 0,C 180,E1 -1976.528,E2 -1976.528} C_VEL
LIN {X 0,Y 580.046,Z 1048.795,A -85,B 0,C 180,E1 -1977.222,E2 -1977.222} C_VEL
LIN {X 0,Y 580.04,Z 1050.592,A -85,B 0,C 180,E1 -1977.917,E2 -1977.917} C_VEL
LIN {X 0,Y 580.044,Z 1051.893,A -85,B 0,C 180,E1 -1978.612,E2 -1978.612} C_VEL
LIN {X 0,Y 580.036,Z 1052.707,A -85,B 0,C 180,E1 -1979.306,E2 -1979.306} C_VEL
LIN {X 0,Y 580.036,Z 1052.996,A -85,B 0,C 180,E1 -1980,E2 -1980} C_VEL
LIN {X 0,Y 580.037,Z 1052.747,A -85,B 0,C 180,E1 -1980.695,E2 -1980.695} C_VEL
LIN {X 0,Y 580.046,Z 1052.014,A -85,B 0,C 180,E1 -1981.389,E2 -1981.389} C_VEL
LIN {X 0,Y 580.041,Z 1050.798,A -85,B 0,C 180,E1 -1982.083,E2 -1982.083} C_VEL
LIN {X 0,Y 580.071,Z 1047.949,A -85,B 0,C 180,E1 -1983.126,E2 -1983.126} C_VEL
LIN {X 0,Y 580.106,Z 1043.849,A -85,B 0,C 180,E1 -1984.169,E2 -1984.169} C_VEL
LIN {X 0,Y 580.091,Z 1038.253,A -85,B 0,C 180,E1 -1985.214,E2 -1985.214} C_VEL
LIN {X 0,Y 580.207,Z 1032.172,A -85,B 0,C 180,E1 -1986.084,E2 -1986.084} C_VEL
LIN {X 0,Y 580.224,Z 1024.503,A -85,B 0,C 180,E1 -1986.957,E2 -1986.957} C_VEL
LIN {X 0,Y 580.276,Z 1015.888,A -85,B 0,C 180,E1 -1987.744,E2 -1987.744} C_VEL
LIN {X 0,Y 580.388,Z 1006.003,A -85,B 0,C 180,E1 -1988.443,E2 -1988.443} C_VEL
LIN {X 0,Y 580.378,Z 996.347,A -85,B 0,C 180,E1 -1988.97,E2 -1988.97} C_VEL
LIN {X 0,Y 580.416,Z 988.121,A -85,B 0,C 180,E1 -1989.321,E2 -1989.321} C_VEL
LIN {X 0,Y 580.458,Z 979.276,A -85,B 0,C 180,E1 -1989.606,E2 -1989.606} C_VEL
LIN {X 0,Y 580.52,Z 970.483,A -85,B 0,C 180,E1 -1989.802,E2 -1989.802} C_VEL
LIN {X 0,Y 580.602,Z 904.705,A -85,B 0,C 180,E1 -1990.633,E2 -1990.633} C_VEL
LIN {X 0,Y 580.471,Z 896.987,A -85,B 0,C 180,E1 -1990.73,E2 -1990.73} C_VEL
LIN {X 0,Y 580.172,Z 894.634,A -85,B 0,C 180,E1 -1990.774,E2 -1990.774} C_VEL
LIN {X 0,Y 580.178,Z 892.53,A -85,B 0,C 180,E1 -1991.219,E2 -1991.219} C_VEL
LIN {X 0,Y 579.512,Z 890.102,A -85,B 0,C 180,E1 -1991.747,E2 -1991.747} C_VEL
LIN {X 0,Y 573.824,Z 882.575,A -85,B 0,C 180,E1 -1993.485,E2 -1993.485} C_VEL
LIN {X 0,Y 573.155,Z 880.165,A -85,B 0,C 180,E1 -1994.022,E2 -1994.022} C_VEL
LIN {X 0,Y 573.303,Z 865.991,A -85,B 0,C 180,E1 -1997.111,E2 -1997.111} C_VEL
LIN {X 0,Y 573.221,Z 863.891,A -85,B 0,C 180,E1 -1997.619,E2 -1997.619} C_VEL
LIN {X 0,Y 573.196,Z 863.891,A -85,B 0,C 180,E1 -2000.079,E2 -2000.079} C_VEL
LIN {X 0,Y 573.186,Z 863.893,A -85,B 0,C 180,E1 -2002.34,E2 -2002.34} C_VEL
LIN {X 0,Y 573.206,Z 863.899,A -85,B 0,C 180,E1 -2005.413,E2 -2005.413} C_VEL
LIN {X 0,Y 573.194,Z 863.893,A -85,B 0,C 180,E1 -2008.018,E2 -2008.018} C_VEL
LIN {X 0,Y 573.202,Z 863.891,A -85,B 0,C 180,E1 -2010.877,E2 -2010.877} C_VEL
LIN {X 0,Y 573.244,Z 863.894,A -85,B 0,C 180,E1 -2013.521,E2 -2013.521} C_VEL
LIN {X 0,Y 573.181,Z 863.899,A -85,B 0,C 180,E1 -2016.055,E2 -2016.055} C_VEL
LIN {X 0,Y 573.214,Z 863.889,A -85,B 0,C 180,E1 -2018.704,E2 -2018.704} C_VEL
LIN {X 0,Y 573.187,Z 863.896,A -85,B 0,C 180,E1 -2021.588,E2 -2021.588} C_VEL
LIN {X 0,Y 573.216,Z 863.896,A -85,B 0,C 180,E1 -2024.336,E2 -2024.336} C_VEL
LIN {X 0,Y 573.206,Z 863.89,A -85,B 0,C 180,E1 -2027.363,E2 -2027.363} C_VEL
LIN {X 0,Y 573.222,Z 863.896,A -85,B 0,C 180,E1 -2030.572,E2 -2030.572} C_VEL
LIN {X 0,Y 573.216,Z 863.891,A -85,B 0,C 180,E1 -2033.075,E2 -2033.075} C_VEL
LIN {X 0,Y 573.243,Z 863.885,A -85,B 0,C 180,E1 -2035.67,E2 -2035.67} C_VEL
LIN {X 0,Y 573.209,Z 863.891,A -85,B 0,C 180,E1 -2038.183,E2 -2038.183} C_VEL
LIN {X 0,Y 573.215,Z 863.896,A -85,B 0,C 180,E1 -2040.631,E2 -2040.631} C_VEL
LIN {X 0,Y 573.197,Z 863.893,A -85,B 0,C 180,E1 -2043.517,E2 -2043.517} C_VEL
LIN {X 0,Y 573.189,Z 863.892,A -85,B 0,C 180,E1 -2046.133,E2 -2046.133} C_VEL
LIN {X 0,Y 573.238,Z 863.896,A -85,B 0,C 180,E1 -2049.173,E2 -2049.173} C_VEL
LIN {X 0,Y 573.194,Z 863.901,A -85,B 0,C 180,E1 -2051.41,E2 -2051.41} C_VEL
LIN {X 0,Y 573.219,Z 863.896,A -85,B 0,C 180,E1 -2053.621,E2 -2053.621} C_VEL
LIN {X 0,Y 573.24,Z 863.891,A -85,B 0,C 180,E1 -2055.806,E2 -2055.806} C_VEL
LIN {X 0,Y 573.231,Z 863.887,A -85,B 0,C 180,E1 -2058.765,E2 -2058.765} C_VEL
LIN {X 0,Y 573.232,Z 863.893,A -85,B 0,C 180,E1 -2061.54,E2 -2061.54} C_VEL
LIN {X 0,Y 573.255,Z 863.887,A -85,B 0,C 180,E1 -2064.372,E2 -2064.372} C_VEL
LIN {X 0,Y 573.309,Z 863.885,A -85,B 0,C 180,E1 -2067.893,E2 -2067.893} C_VEL
LIN {X 0,Y 573.319,Z 863.884,A -85,B 0,C 180,E1 -2070,E2 -2070} C_VEL
LIN {X 0,Y 573.272,Z 863.884,A -85,B 0,C 180,E1 -2072.811,E2 -2072.811} C_VEL
LIN {X 0,Y 573.25,Z 863.885,A -85,B 0,C 180,E1 -2075.629,E2 -2075.629} C_VEL
LIN {X 0,Y 573.233,Z 863.897,A -85,B 0,C 180,E1 -2078.46,E2 -2078.46} C_VEL
LIN {X 0,Y 573.238,Z 863.887,A -85,B 0,C 180,E1 -2081.313,E2 -2081.313} C_VEL
LIN {X 0,Y 573.229,Z 863.891,A -85,B 0,C 180,E1 -2084.401,E2 -2084.401} C_VEL
LIN {X 0,Y 573.222,Z 863.895,A -85,B 0,C 180,E1 -2087.113,E2 -2087.113} C_VEL
LIN {X 0,Y 573.197,Z 863.891,A -85,B 0,C 180,E1 -2090.079,E2 -2090.079} C_VEL
LIN {X 0,Y 573.186,Z 863.892,A -85,B 0,C 180,E1 -2092.34,E2 -2092.34} C_VEL
LIN {X 0,Y 573.193,Z 863.896,A -85,B 0,C 180,E1 -2094.86,E2 -2094.86} C_VEL
LIN {X 0,Y 573.189,Z 863.897,A -85,B 0,C 180,E1 -2096.979,E2 -2096.979} C_VEL
LIN {X 0,Y 573.201,Z 863.901,A -85,B 0,C 180,E1 -2099.479,E2 -2099.479} C_VEL
LIN {X 0,Y 573.197,Z 863.892,A -85,B 0,C 180,E1 -2102.218,E2 -2102.218} C_VEL
LIN {X 0,Y 573.217,Z 863.888,A -85,B 0,C 180,E1 -2104.768,E2 -2104.768} C_VEL
LIN {X 0,Y 573.19,Z 863.903,A -85,B 0,C 180,E1 -2107.811,E2 -2107.811} C_VEL
LIN {X 0,Y 573.204,Z 863.892,A -85,B 0,C 180,E1 -2110.529,E2 -2110.529} C_VEL
LIN {X 0,Y 573.191,Z 863.893,A -85,B 0,C 180,E1 -2113.364,E2 -2113.364} C_VEL
LIN {X 0,Y 573.195,Z 863.9,A -85,B 0,C 180,E1 -2116.337,E2 -2116.337} C_VEL
LIN {X 0,Y 573.187,Z 863.899,A -85,B 0,C 180,E1 -2118.538,E2 -2118.538} C_VEL
LIN {X 0,Y 573.176,Z 863.893,A -85,B 0,C 180,E1 -2121.293,E2 -2121.293} C_VEL
LIN {X 0,Y 573.183,Z 863.895,A -85,B 0,C 180,E1 -2124.023,E2 -2124.023} C_VEL
LIN {X 0,Y 573.226,Z 863.896,A -85,B 0,C 180,E1 -2126.514,E2 -2126.514} C_VEL
LIN {X 0,Y 573.204,Z 863.895,A -85,B 0,C 180,E1 -2129.123,E2 -2129.123} C_VEL
LIN {X 0,Y 573.196,Z 863.891,A -85,B 0,C 180,E1 -2131.982,E2 -2131.982} C_VEL
LIN {X 0,Y 573.199,Z 863.894,A -85,B 0,C 180,E1 -2134.587,E2 -2134.587} C_VEL
LIN {X 0,Y 573.207,Z 863.892,A -85,B 0,C 180,E1 -2137.661,E2 -2137.661} C_VEL
LIN {X 0,Y 573.2,Z 863.891,A -85,B 0,C 180,E1 -2139.921,E2 -2139.921} C_VEL
LIN {X 0,Y 573.217,Z 863.893,A -85,B 0,C 180,E1 -2143.006,E2 -2143.006} C_VEL
LIN {X 0,Y 573.225,Z 863.893,A -85,B 0,C 180,E1 -2145.805,E2 -2145.805} C_VEL
LIN {X 0,Y 573.23,Z 863.887,A -85,B 0,C 180,E1 -2148.764,E2 -2148.764} C_VEL
LIN {X 0,Y 573.231,Z 863.894,A -85,B 0,C 180,E1 -2151.539,E2 -2151.539} C_VEL
LIN {X 0,Y 573.253,Z 863.887,A -85,B 0,C 180,E1 -2154.371,E2 -2154.371} C_VEL
LIN {X 0,Y 573.308,Z 863.886,A -85,B 0,C 180,E1 -2157.892,E2 -2157.892} C_VEL
LIN {X 0,Y 573.317,Z 863.885,A -85,B 0,C 180,E1 -2160,E2 -2160} C_VEL
LIN {X 0,Y 573.269,Z 863.884,A -85,B 0,C 180,E1 -2162.81,E2 -2162.81} C_VEL
LIN {X 0,Y 573.248,Z 863.885,A -85,B 0,C 180,E1 -2165.628,E2 -2165.628} C_VEL
LIN {X 0,Y 573.231,Z 863.897,A -85,B 0,C 180,E1 -2168.46,E2 -2168.46} C_VEL
LIN {X 0,Y 573.235,Z 863.887,A -85,B 0,C 180,E1 -2171.312,E2 -2171.312} C_VEL
LIN {X 0,Y 573.247,Z 863.889,A -85,B 0,C 180,E1 -2174.409,E2 -2174.409} C_VEL
LIN {X 0,Y 573.219,Z 863.895,A -85,B 0,C 180,E1 -2177.113,E2 -2177.113} C_VEL
LIN {X 0,Y 573.194,Z 863.891,A -85,B 0,C 180,E1 -2180.078,E2 -2180.078} C_VEL
LIN {X 0,Y 573.184,Z 863.893,A -85,B 0,C 180,E1 -2182.34,E2 -2182.34} C_VEL
LIN {X 0,Y 573.189,Z 863.896,A -85,B 0,C 180,E1 -2184.86,E2 -2184.86} C_VEL
LIN {X 0,Y 573.185,Z 863.897,A -85,B 0,C 180,E1 -2186.979,E2 -2186.979} C_VEL
LIN {X 0,Y 573.197,Z 863.901,A -85,B 0,C 180,E1 -2189.478,E2 -2189.478} C_VEL
LIN {X 0,Y 573.193,Z 863.892,A -85,B 0,C 180,E1 -2192.218,E2 -2192.218} C_VEL
LIN {X 0,Y 573.213,Z 863.889,A -85,B 0,C 180,E1 -2194.768,E2 -2194.768} C_VEL
LIN {X 0,Y 573.193,Z 863.902,A -85,B 0,C 180,E1 -2197.811,E2 -2197.811} C_VEL
LIN {X 0,Y 573.2,Z 863.892,A -85,B 0,C 180,E1 -2200.529,E2 -2200.529} C_VEL
LIN {X 0,Y 573.19,Z 863.893,A -85,B 0,C 180,E1 -2203.363,E2 -2203.363} C_VEL
LIN {X 0,Y 573.192,Z 863.9,A -85,B 0,C 180,E1 -2206.336,E2 -2206.336} C_VEL
LIN {X 0,Y 573.183,Z 863.899,A -85,B 0,C 180,E1 -2208.538,E2 -2208.538} C_VEL
LIN {X 0,Y 573.173,Z 863.894,A -85,B 0,C 180,E1 -2211.293,E2 -2211.293} C_VEL
LIN {X 0,Y 573.179,Z 863.896,A -85,B 0,C 180,E1 -2214.023,E2 -2214.023} C_VEL
LIN {X 0,Y 573.221,Z 863.897,A -85,B 0,C 180,E1 -2216.514,E2 -2216.514} C_VEL
LIN {X 0,Y 573.2,Z 863.895,A -85,B 0,C 180,E1 -2219.123,E2 -2219.123} C_VEL
LIN {X 0,Y 573.192,Z 863.891,A -85,B 0,C 180,E1 -2221.982,E2 -2221.982} C_VEL
LIN {X 0,Y 573.195,Z 863.897,A -85,B 0,C 180,E1 -2224.587,E2 -2224.587} C_VEL
LIN {X 0,Y 573.22,Z 863.896,A -85,B 0,C 180,E1 -2227.661,E2 -2227.661} C_VEL
LIN {X 0,Y 573.255,Z 864.154,A -85,B 0,C 180,E1 -2227.852,E2 -2227.852} C_VEL
LIN {X 0,Y 573.76,Z 868.328,A -85,B 0,C 180,E1 -2228.579,E2 -2228.579} C_VEL
LIN {X 0,Y 573.556,Z 885.369,A -85,B 0,C 180,E1 -2231.422,E2 -2231.422} C_VEL
LIN {X 0,Y 573.397,Z 902.118,A -85,B 0,C 180,E1 -2234.174,E2 -2234.174} C_VEL
LIN {X 0,Y 573.262,Z 919.983,A -85,B 0,C 180,E1 -2237.071,E2 -2237.071} C_VEL
LIN {X 0,Y 573.172,Z 932.757,A -85,B 0,C 180,E1 -2239.123,E2 -2239.123} C_VEL
LIN {X 0,Y 573.65,Z 938.219,A -85,B 0,C 180,E1 -2239.201,E2 -2239.201} C_VEL
LIN {X 0,Y 573.542,Z 1009.13,A -85,B 0,C 180,E1 -2240.1,E2 -2240.1} C_VEL
LIN {X 0,Y 573.495,Z 1018.407,A -85,B 0,C 180,E1 -2240.299,E2 -2240.299} C_VEL
LIN {X 0,Y 573.443,Z 1026.887,A -85,B 0,C 180,E1 -2240.565,E2 -2240.565} C_VEL
LIN {X 0,Y 573.393,Z 1035.394,A -85,B 0,C 180,E1 -2240.92,E2 -2240.92} C_VEL
LIN {X 0,Y 573.366,Z 1043.725,A -85,B 0,C 180,E1 -2241.364,E2 -2241.364} C_VEL
LIN {X 0,Y 573.256,Z 1051.763,A -85,B 0,C 180,E1 -2241.895,E2 -2241.895} C_VEL
LIN {X 0,Y 573.187,Z 1059.414,A -85,B 0,C 180,E1 -2242.514,E2 -2242.514} C_VEL
LIN {X 0,Y 573.155,Z 1067.545,A -85,B 0,C 180,E1 -2243.322,E2 -2243.322} C_VEL
